LIN {X 0,Y 269.686,Z 884.674,A -85,B 0,C 180,E1 -12883.072,E2 -12883.072} C_VEL
LIN {X 0,Y 271.934,Z 878.624,A -85,B 0,C 180,E1 -12886.887,E2 -12886.887} C_VEL
LIN {X 0,Y 274.765,Z 871.156,A -85,B 0,C 180,E1 -12890.448,E2 -12890.448} C_VEL
LIN {X 0,Y 278.331,Z 861.736,A -85,B 0,C 180,E1 -12893.95,E2 -12893.95} C_VEL
LIN {X 0,Y 282.374,Z 850.757,A -85,B 0,C 180,E1 -12897.18,E2 -12897.18} C_VEL
LIN {X 0,Y 286.714,Z 838.141,A -85,B 0,C 180,E1 -12900.144,E2 -12900.144} C_VEL
LIN {X 0,Y 291.068,Z 824.299,A -85,B 0,C 180,E1 -12902.755,E2 -12902.755} C_VEL
LIN {X 0,Y 295.08,Z 810.044,A -85,B 0,C 180,E1 -12904.936,E2 -12904.936} C_VEL
LIN {X 0,Y 298.861,Z 794.399,A -85,B 0,C 180,E1 -12906.875,E2 -12906.875} C_VEL
LIN {X 0,Y 302.134,Z 778.251,A -85,B 0,C 180,E1 -12908.474,E2 -12908.474} C_VEL
LIN {X 0,Y 304.902,Z 760.982,A -85,B 0,C 180,E1 -12909.813,E2 -12909.813} C_VEL
LIN {X 0,Y 306.977,Z 742.738,A -85,B 0,C 180,E1 -12910.881,E2 -12910.881} C_VEL
LIN {X 0,Y 308.237,Z 723.755,A -85,B 0,C 180,E1 -12911.658,E2 -12911.658} C_VEL
LIN {X 0,Y 309.895,Z 682.456,A -85,B 0,C 180,E1 -12912.705,E2 -12912.705} C_VEL
LIN {X 0,Y 310.726,Z 666.212,A -85,B 0,C 180,E1 -12913.069,E2 -12913.069} C_VEL
LIN {X 0,Y 310.408,Z 658.622,A -85,B 0,C 180,E1 -12913.367,E2 -12913.367} C_VEL
LIN {X 0,Y 307.038,Z 638.78,A -85,B 0,C 180,E1 -12914.632,E2 -12914.632} C_VEL
LIN {X 0,Y 306.867,Z 632.255,A -85,B 0,C 180,E1 -12914.879,E2 -12914.879} C_VEL
LIN {X 0,Y 310.629,Z 562.408,A -85,B 0,C 180,E1 -12916.462,E2 -12916.462} C_VEL
LIN {X 0,Y 306.876,Z 565.093,A -85,B 0,C 180,E1 -12917.138,E2 -12917.138} C_VEL
LIN {X 0,Y 301.533,Z 573.563,A -85,B 0,C 180,E1 -12917.98,E2 -12917.98} C_VEL
LIN {X 0,Y 297.455,Z 578.086,A -85,B 0,C 180,E1 -12918.725,E2 -12918.725} C_VEL
LIN {X 0,Y 295.264,Z 579.155,A -85,B 0,C 180,E1 -12919.189,E2 -12919.189} C_VEL
LIN {X 0,Y 294.567,Z 579.193,A -85,B 0,C 180,E1 -12919.371,E2 -12919.371} C_VEL
LIN {X 0,Y 288.038,Z 619.211,A -85,B 0,C 180,E1 -12923.908,E2 -12923.908} C_VEL
LIN {X 0,Y 288.137,Z 629.093,A -85,B 0,C 180,E1 -12924.423,E2 -12924.423} C_VEL
LIN {X 0,Y 279.258,Z 720.889,A -85,B 0,C 180,E1 -12928.189,E2 -12928.189} C_VEL
LIN {X 0,Y 275.539,Z 766.557,A -85,B 0,C 180,E1 -12930.346,E2 -12930.346} C_VEL
LIN {X 0,Y 274.092,Z 785.081,A -85,B 0,C 180,E1 -12931.514,E2 -12931.514} C_VEL
LIN {X 0,Y 272.218,Z 802.313,A -85,B 0,C 180,E1 -12933.023,E2 -12933.023} C_VEL
LIN {X 0,Y 270.16,Z 818.126,A -85,B 0,C 180,E1 -12934.81,E2 -12934.81} C_VEL
LIN {X 0,Y 267.771,Z 834.431,A -85,B 0,C 180,E1 -12937.148,E2 -12937.148} C_VEL
LIN {X 0,Y 265.418,Z 849.249,A -85,B 0,C 180,E1 -12939.836,E2 -12939.836} C_VEL
LIN {X 0,Y 263.474,Z 861.324,A -85,B 0,C 180,E1 -12942.554,E2 -12942.554} C_VEL
LIN {X 0,Y 261.789,Z 872.401,A -85,B 0,C 180,E1 -12945.625,E2 -12945.625} C_VEL
LIN {X 0,Y 260.5,Z 881.93,A -85,B 0,C 180,E1 -12948.935,E2 -12948.935} C_VEL
LIN {X 0,Y 259.751,Z 889.559,A -85,B 0,C 180,E1 -12952.257,E2 -12952.257} C_VEL
LIN {X 0,Y 259.465,Z 896.044,A -85,B 0,C 180,E1 -12956.022,E2 -12956.022} C_VEL
LIN {X 0,Y 259.712,Z 900.395,A -85,B 0,C 180,E1 -12959.558,E2 -12959.558} C_VEL
LIN {X 0,Y 260.599,Z 903.408,A -85,B 0,C 180,E1 -12963.519,E2 -12963.519} C_VEL
LIN {X 0,Y 262.216,Z 904.421,A -85,B 0,C 180,E1 -12967.448,E2 -12967.448} C_VEL
LIN {X 0,Y 264.534,Z 903.668,A -85,B 0,C 180,E1 -12971.114,E2 -12971.114} C_VEL
LIN {X 0,Y 267.932,Z 901.106,A -85,B 0,C 180,E1 -12974.921,E2 -12974.921} C_VEL
LIN {X 0,Y 272.584,Z 896.369,A -85,B 0,C 180,E1 -12978.831,E2 -12978.831} C_VEL
LIN {X 0,Y 278.094,Z 889.924,A -85,B 0,C 180,E1 -12982.402,E2 -12982.402} C_VEL
LIN {X 0,Y 284.71,Z 881.473,A -85,B 0,C 180,E1 -12985.815,E2 -12985.815} C_VEL
LIN {X 0,Y 292.053,Z 871.644,A -85,B 0,C 180,E1 -12988.863,E2 -12988.863} C_VEL
LIN {X 0,Y 301.107,Z 859.274,A -85,B 0,C 180,E1 -12991.868,E2 -12991.868} C_VEL
LIN {X 0,Y 311.714,Z 844.887,A -85,B 0,C 180,E1 -12994.593,E2 -12994.593} C_VEL
LIN {X 0,Y 322.865,Z 830.154,A -85,B 0,C 180,E1 -12996.789,E2 -12996.789} C_VEL
LIN {X 0,Y 309.588,Z 851.693,A -85,B 0,C 180,E1 -12999.476,E2 -12999.476} C_VEL
LIN {X 0,Y 296.509,Z 873.71,A -85,B 0,C 180,E1 -13002.966,E2 -13002.966} C_VEL
LIN {X 0,Y 284.849,Z 895.114,A -85,B 0,C 180,E1 -13007.19,E2 -13007.19} C_VEL
LIN {X 0,Y 275.724,Z 913.791,A -85,B 0,C 180,E1 -13011.676,E2 -13011.676} C_VEL
LIN {X 0,Y 268.77,Z 929.861,A -85,B 0,C 180,E1 -13016.337,E2 -13016.337} C_VEL
LIN {X 0,Y 263.613,Z 943.776,A -85,B 0,C 180,E1 -13021.203,E2 -13021.203} C_VEL
LIN {X 0,Y 260.112,Z 955.453,A -85,B 0,C 180,E1 -13026.195,E2 -13026.195} C_VEL
LIN {X 0,Y 258.142,Z 964.49,A -85,B 0,C 180,E1 -13031.012,E2 -13031.012} C_VEL
LIN {X 0,Y 257.314,Z 970.99,A -85,B 0,C 180,E1 -13035.369,E2 -13035.369} C_VEL
LIN {X 0,Y 257.198,Z 975.8,A -85,B 0,C 180,E1 -13039.698,E2 -13039.698} C_VEL
LIN {X 0,Y 257.448,Z 979.006,A -85,B 0,C 180,E1 -13043.98,E2 -13043.98} C_VEL
LIN {X 0,Y 257.684,Z 980.43,A -85,B 0,C 180,E1 -13047.776,E2 -13047.776} C_VEL
LIN {X 0,Y 257.745,Z 980.427,A -85,B 0,C 180,E1 -13051.555,E2 -13051.555} C_VEL
LIN {X 0,Y 257.572,Z 979.005,A -85,B 0,C 180,E1 -13055.345,E2 -13055.345} C_VEL
LIN {X 0,Y 257.333,Z 975.954,A -85,B 0,C 180,E1 -13059.391,E2 -13059.391} C_VEL
LIN {X 0,Y 257.405,Z 971.221,A -85,B 0,C 180,E1 -13063.477,E2 -13063.477} C_VEL
LIN {X 0,Y 257.989,Z 964.85,A -85,B 0,C 180,E1 -13067.595,E2 -13067.595} C_VEL
LIN {X 0,Y 259.502,Z 955.672,A -85,B 0,C 180,E1 -13072.184,E2 -13072.184} C_VEL
LIN {X 0,Y 261.93,Z 944.738,A -85,B 0,C 180,E1 -13076.526,E2 -13076.526} C_VEL
LIN {X 0,Y 265.436,Z 931.412,A -85,B 0,C 180,E1 -13080.816,E2 -13080.816} C_VEL
LIN {X 0,Y 269.811,Z 916.263,A -85,B 0,C 180,E1 -13084.798,E2 -13084.798} C_VEL
LIN {X 0,Y 274.746,Z 899.855,A -85,B 0,C 180,E1 -13088.351,E2 -13088.351} C_VEL
LIN {X 0,Y 280.04,Z 882.42,A -85,B 0,C 180,E1 -13091.476,E2 -13091.476} C_VEL
LIN {X 0,Y 285.407,Z 864.061,A -85,B 0,C 180,E1 -13094.198,E2 -13094.198} C_VEL
LIN {X 0,Y 291.22,Z 843.632,A -85,B 0,C 180,E1 -13096.707,E2 -13096.707} C_VEL
LIN {X 0,Y 296.821,Z 822.506,A -85,B 0,C 180,E1 -13098.839,E2 -13098.839} C_VEL
LIN {X 0,Y 302.079,Z 800.854,A -85,B 0,C 180,E1 -13100.611,E2 -13100.611} C_VEL
LIN {X 0,Y 307.337,Z 776.523,A -85,B 0,C 180,E1 -13102.16,E2 -13102.16} C_VEL
LIN {X 0,Y 311.674,Z 752.148,A -85,B 0,C 180,E1 -13103.33,E2 -13103.33} C_VEL
LIN {X 0,Y 314.616,Z 728.619,A -85,B 0,C 180,E1 -13104.182,E2 -13104.182} C_VEL
LIN {X 0,Y 318.188,Z 703.693,A -85,B 0,C 180,E1 -13104.767,E2 -13104.767} C_VEL
LIN {X 0,Y 319.534,Z 697.27,A -85,B 0,C 180,E1 -13104.911,E2 -13104.911} C_VEL
LIN {X 0,Y 333.437,Z 667.218,A -85,B 0,C 180,E1 -13106.472,E2 -13106.472} C_VEL
LIN {X 0,Y 344.021,Z 646.575,A -85,B 0,C 180,E1 -13107.351,E2 -13107.351} C_VEL
LIN {X 0,Y 339.833,Z 627.474,A -85,B 0,C 180,E1 -13110.221,E2 -13110.221} C_VEL
LIN {X 0,Y 337.763,Z 606.391,A -85,B 0,C 180,E1 -13113.165,E2 -13113.165} C_VEL
LIN {X 0,Y 338.071,Z 583.429,A -85,B 0,C 180,E1 -13116.098,E2 -13116.098} C_VEL
LIN {X 0,Y 340.611,Z 559.678,A -85,B 0,C 180,E1 -13118.835,E2 -13118.835} C_VEL
LIN {X 0,Y 342.754,Z 547.466,A -85,B 0,C 180,E1 -13120.133,E2 -13120.133} C_VEL
LIN {X 0,Y 334.601,Z 531.23,A -85,B 0,C 180,E1 -13124.222,E2 -13124.222} C_VEL
LIN {X 0,Y 325.953,Z 514.792,A -85,B 0,C 180,E1 -13128.858,E2 -13128.858} C_VEL
LIN {X 0,Y 318.261,Z 500.611,A -85,B 0,C 180,E1 -13133.325,E2 -13133.325} C_VEL
LIN {X 0,Y 310.915,Z 487.26,A -85,B 0,C 180,E1 -13137.973,E2 -13137.973} C_VEL
LIN {X 0,Y 304.028,Z 475.288,A -85,B 0,C 180,E1 -13142.639,E2 -13142.639} C_VEL
LIN {X 0,Y 298.834,Z 466.349,A -85,B 0,C 180,E1 -13146.427,E2 -13146.427} C_VEL
LIN {X 0,Y 295.334,Z 460.31,A -85,B 0,C 180,E1 -13149.156,E2 -13149.156} C_VEL
LIN {X 0,Y 292.811,Z 455.963,A -85,B 0,C 180,E1 -13151.224,E2 -13151.224} C_VEL
LIN {X 0,Y 290.37,Z 451.67,A -85,B 0,C 180,E1 -13153.339,E2 -13153.339} C_VEL
LIN {X 0,Y 287.246,Z 446.365,A -85,B 0,C 180,E1 -13156.115,E2 -13156.115} C_VEL
LIN {X 0,Y 284.576,Z 441.72,A -85,B 0,C 180,E1 -13158.647,E2 -13158.647} C_VEL
LIN {X 0,Y 281.501,Z 436.433,A -85,B 0,C 180,E1 -13161.788,E2 -13161.788} C_VEL
LIN {X 0,Y 285.523,Z 436.484,A -85,B 0,C 180,E1 -13163.749,E2 -13163.749} C_VEL
LIN {X 0,Y 288.01,Z 440.52,A -85,B 0,C 180,E1 -13165.499,E2 -13165.499} C_VEL
LIN {X 0,Y 292.612,Z 448.472,A -85,B 0,C 180,E1 -13168.469,E2 -13168.469} C_VEL
LIN {X 0,Y 298.931,Z 460.913,A -85,B 0,C 180,E1 -13172.356,E2 -13172.356} C_VEL
LIN {X 0,Y 305.142,Z 474.876,A -85,B 0,C 180,E1 -13175.969,E2 -13175.969} C_VEL
LIN {X 0,Y 310.504,Z 488.843,A -85,B 0,C 180,E1 -13179.016,E2 -13179.016} C_VEL
LIN {X 0,Y 313.865,Z 499.241,A -85,B 0,C 180,E1 -13180.976,E2 -13180.976} C_VEL
LIN {X 0,Y 312.333,Z 517.888,A -85,B 0,C 180,E1 -13182.511,E2 -13182.511} C_VEL
LIN {X 0,Y 312.75,Z 525.28,A -85,B 0,C 180,E1 -13182.848,E2 -13182.848} C_VEL
LIN {X 0,Y 302.694,Z 713.065,A -85,B 0,C 180,E1 -13187.105,E2 -13187.105} C_VEL
LIN {X 0,Y 301.697,Z 734.677,A -85,B 0,C 180,E1 -13187.816,E2 -13187.816} C_VEL
LIN {X 0,Y 299.958,Z 753.181,A -85,B 0,C 180,E1 -13188.749,E2 -13188.749} C_VEL
LIN {X 0,Y 297.437,Z 770.891,A -85,B 0,C 180,E1 -13189.967,E2 -13189.967} C_VEL
LIN {X 0,Y 294.321,Z 787.313,A -85,B 0,C 180,E1 -13191.425,E2 -13191.425} C_VEL
LIN {X 0,Y 290.622,Z 803.379,A -85,B 0,C 180,E1 -13193.229,E2 -13193.229} C_VEL
LIN {X 0,Y 286.527,Z 818.441,A -85,B 0,C 180,E1 -13195.334,E2 -13195.334} C_VEL
LIN {X 0,Y 282.137,Z 832.541,A -85,B 0,C 180,E1 -13197.768,E2 -13197.768} C_VEL
LIN {X 0,Y 277.8,Z 845.153,A -85,B 0,C 180,E1 -13200.457,E2 -13200.457} C_VEL
LIN {X 0,Y 273.502,Z 856.753,A -85,B 0,C 180,E1 -13203.513,E2 -13203.513} C_VEL
LIN {X 0,Y 269.379,Z 867.277,A -85,B 0,C 180,E1 -13207.002,E2 -13207.002} C_VEL
LIN {X 0,Y 265.876,Z 876.028,A -85,B 0,C 180,E1 -13210.722,E2 -13210.722} C_VEL
LIN {X 0,Y 263.109,Z 882.968,A -85,B 0,C 180,E1 -13214.574,E2 -13214.574} C_VEL
LIN {X 0,Y 261.045,Z 888.364,A -85,B 0,C 180,E1 -13218.679,E2 -13218.679} C_VEL
LIN {X 0,Y 259.745,Z 892.055,A -85,B 0,C 180,E1 -13222.925,E2 -13222.925} C_VEL
LIN {X 0,Y 259.111,Z 893.998,A -85,B 0,C 180,E1 -13227.125,E2 -13227.125} C_VEL
LIN {X 0,Y 259.011,Z 894.319,A -85,B 0,C 180,E1 -13231.328,E2 -13231.328} C_VEL
LIN {X 0,Y 259.438,Z 893.029,A -85,B 0,C 180,E1 -13235.53,E2 -13235.53} C_VEL
LIN {X 0,Y 260.445,Z 890.085,A -85,B 0,C 180,E1 -13239.726,E2 -13239.726} C_VEL
LIN {X 0,Y 262.204,Z 885.377,A -85,B 0,C 180,E1 -13243.901,E2 -13243.901} C_VEL
LIN {X 0,Y 264.702,Z 879.086,A -85,B 0,C 180,E1 -13247.845,E2 -13247.845} C_VEL
LIN {X 0,Y 267.966,Z 870.939,A -85,B 0,C 180,E1 -13251.679,E2 -13251.679} C_VEL
LIN {X 0,Y 271.854,Z 861.1,A -85,B 0,C 180,E1 -13255.255,E2 -13255.255} C_VEL
LIN {X 0,Y 275.924,Z 850.446,A -85,B 0,C 180,E1 -13258.341,E2 -13258.341} C_VEL
LIN {X 0,Y 280.217,Z 838.43,A -85,B 0,C 180,E1 -13261.158,E2 -13261.158} C_VEL
LIN {X 0,Y 284.623,Z 824.969,A -85,B 0,C 180,E1 -13263.714,E2 -13263.714} C_VEL
LIN {X 0,Y 288.821,Z 810.587,A -85,B 0,C 180,E1 -13265.93,E2 -13265.93} C_VEL
LIN {X 0,Y 292.63,Z 795.395,A -85,B 0,C 180,E1 -13267.83,E2 -13267.83} C_VEL
LIN {X 0,Y 295.986,Z 779.481,A -85,B 0,C 180,E1 -13269.426,E2 -13269.426} C_VEL
LIN {X 0,Y 298.869,Z 762.198,A -85,B 0,C 180,E1 -13270.784,E2 -13270.784} C_VEL
LIN {X 0,Y 301.034,Z 743.929,A -85,B 0,C 180,E1 -13271.867,E2 -13271.867} C_VEL
LIN {X 0,Y 302.358,Z 724.895,A -85,B 0,C 180,E1 -13272.657,E2 -13272.657} C_VEL
LIN {X 0,Y 304.093,Z 683.595,A -85,B 0,C 180,E1 -13273.721,E2 -13273.721} C_VEL
LIN {X 0,Y 306.867,Z 632.255,A -85,B 0,C 180,E1 -13274.879,E2 -13274.879} C_VEL
LIN {X 0,Y 306.592,Z 624.667,A -85,B 0,C 180,E1 -13275.183,E2 -13275.183} C_VEL
LIN {X 0,Y 303.427,Z 604.831,A -85,B 0,C 180,E1 -13276.486,E2 -13276.486} C_VEL
LIN {X 0,Y 303.291,Z 598.308,A -85,B 0,C 180,E1 -13276.739,E2 -13276.739} C_VEL
LIN {X 0,Y 304.281,Z 579.807,A -85,B 0,C 180,E1 -13277.172,E2 -13277.172} C_VEL
LIN {X 0,Y 299.607,Z 584.811,A -85,B 0,C 180,E1 -13278,E2 -13278} C_VEL
LIN {X 0,Y 296.722,Z 586.907,A -85,B 0,C 180,E1 -13278.568,E2 -13278.568} C_VEL
LIN {X 0,Y 291.301,Z 595.969,A -85,B 0,C 180,E1 -13279.489,E2 -13279.489} C_VEL
LIN {X 0,Y 287.307,Z 600.801,A -85,B 0,C 180,E1 -13280.274,E2 -13280.274} C_VEL
LIN {X 0,Y 284.901,Z 602.253,A -85,B 0,C 180,E1 -13280.823,E2 -13280.823} C_VEL
LIN {X 0,Y 284.207,Z 602.229,A -85,B 0,C 180,E1 -13281.011,E2 -13281.011} C_VEL
LIN {X 0,Y 281.343,Z 620.048,A -85,B 0,C 180,E1 -13283.037,E2 -13283.037} C_VEL
LIN {X 0,Y 281.385,Z 629.859,A -85,B 0,C 180,E1 -13283.565,E2 -13283.565} C_VEL
LIN {X 0,Y 271.871,Z 723.942,A -85,B 0,C 180,E1 -13287.555,E2 -13287.555} C_VEL
LIN {X 0,Y 268.167,Z 767.49,A -85,B 0,C 180,E1 -13289.708,E2 -13289.708} C_VEL
LIN {X 0,Y 266.603,Z 786.293,A -85,B 0,C 180,E1 -13290.943,E2 -13290.943} C_VEL
LIN {X 0,Y 264.596,Z 804.008,A -85,B 0,C 180,E1 -13292.547,E2 -13292.547} C_VEL
LIN {X 0,Y 262.469,Z 819.69,A -85,B 0,C 180,E1 -13294.381,E2 -13294.381} C_VEL
LIN {X 0,Y 260.11,Z 835.238,A -85,B 0,C 180,E1 -13296.675,E2 -13296.675} C_VEL
LIN {X 0,Y 257.753,Z 849.521,A -85,B 0,C 180,E1 -13299.328,E2 -13299.328} C_VEL
LIN {X 0,Y 255.647,Z 862.213,A -85,B 0,C 180,E1 -13302.237,E2 -13302.237} C_VEL
LIN {X 0,Y 253.798,Z 874.116,A -85,B 0,C 180,E1 -13305.629,E2 -13305.629} C_VEL
LIN {X 0,Y 252.446,Z 884.164,A -85,B 0,C 180,E1 -13309.271,E2 -13309.271} C_VEL
LIN {X 0,Y 251.737,Z 891.577,A -85,B 0,C 180,E1 -13312.697,E2 -13312.697} C_VEL
LIN {X 0,Y 251.545,Z 897.997,A -85,B 0,C 180,E1 -13316.581,E2 -13316.581} C_VEL
LIN {X 0,Y 251.945,Z 902.424,A -85,B 0,C 180,E1 -13320.454,E2 -13320.454} C_VEL
LIN {X 0,Y 252.97,Z 905.133,A -85,B 0,C 180,E1 -13324.306,E2 -13324.306} C_VEL
LIN {X 0,Y 254.835,Z 906.14,A -85,B 0,C 180,E1 -13328.347,E2 -13328.347} C_VEL
LIN {X 0,Y 257.823,Z 905.177,A -85,B 0,C 180,E1 -13332.542,E2 -13332.542} C_VEL
LIN {X 0,Y 261.946,Z 902.204,A -85,B 0,C 180,E1 -13336.635,E2 -13336.635} C_VEL
LIN {X 0,Y 267.259,Z 897.237,A -85,B 0,C 180,E1 -13340.589,E2 -13340.589} C_VEL
LIN {X 0,Y 273.829,Z 890.233,A -85,B 0,C 180,E1 -13344.368,E2 -13344.368} C_VEL
LIN {X 0,Y 281.246,Z 881.626,A -85,B 0,C 180,E1 -13347.756,E2 -13347.756} C_VEL
LIN {X 0,Y 290.467,Z 870.573,A -85,B 0,C 180,E1 -13351.086,E2 -13351.086} C_VEL
LIN {X 0,Y 301.272,Z 857.503,A -85,B 0,C 180,E1 -13354.116,E2 -13354.116} C_VEL
LIN {X 0,Y 313.457,Z 843.065,A -85,B 0,C 180,E1 -13356.732,E2 -13356.732} C_VEL
LIN {X 0,Y 299.81,Z 863.023,A -85,B 0,C 180,E1 -13359.611,E2 -13359.611} C_VEL
LIN {X 0,Y 286.869,Z 883.051,A -85,B 0,C 180,E1 -13363.242,E2 -13363.242} C_VEL
LIN {X 0,Y 275.073,Z 903.185,A -85,B 0,C 180,E1 -13367.742,E2 -13367.742} C_VEL
LIN {X 0,Y 265.677,Z 921.336,A -85,B 0,C 180,E1 -13372.705,E2 -13372.705} C_VEL
LIN {X 0,Y 258.843,Z 936.59,A -85,B 0,C 180,E1 -13377.786,E2 -13377.786} C_VEL
LIN {X 0,Y 253.997,Z 949.606,A -85,B 0,C 180,E1 -13383.082,E2 -13383.082} C_VEL
LIN {X 0,Y 250.974,Z 960.274,A -85,B 0,C 180,E1 -13388.498,E2 -13388.498} C_VEL
LIN {X 0,Y 249.639,Z 967.637,A -85,B 0,C 180,E1 -13393.239,E2 -13393.239} C_VEL
LIN {X 0,Y 249.22,Z 973.262,A -85,B 0,C 180,E1 -13397.958,E2 -13397.958} C_VEL
LIN {X 0,Y 249.399,Z 976.902,A -85,B 0,C 180,E1 -13402.397,E2 -13402.397} C_VEL
LIN {X 0,Y 249.717,Z 978.754,A -85,B 0,C 180,E1 -13406.326,E2 -13406.326} C_VEL
LIN {X 0,Y 249.877,Z 979.213,A -85,B 0,C 180,E1 -13410.229,E2 -13410.229} C_VEL
LIN {X 0,Y 249.769,Z 978.324,A -85,B 0,C 180,E1 -13413.902,E2 -13413.902} C_VEL
LIN {X 0,Y 249.523,Z 975.953,A -85,B 0,C 180,E1 -13417.83,E2 -13417.83} C_VEL
LIN {X 0,Y 249.426,Z 971.821,A -85,B 0,C 180,E1 -13422.031,E2 -13422.031} C_VEL
LIN {X 0,Y 249.806,Z 966.033,A -85,B 0,C 180,E1 -13426.27,E2 -13426.27} C_VEL
LIN {X 0,Y 250.953,Z 958.015,A -85,B 0,C 180,E1 -13430.768,E2 -13430.768} C_VEL
LIN {X 0,Y 253.071,Z 947.881,A -85,B 0,C 180,E1 -13435.257,E2 -13435.257} C_VEL
LIN {X 0,Y 256.087,Z 936.144,A -85,B 0,C 180,E1 -13439.468,E2 -13439.468} C_VEL
LIN {X 0,Y 259.96,Z 922.745,A -85,B 0,C 180,E1 -13443.424,E2 -13443.424} C_VEL
LIN {X 0,Y 264.675,Z 907.329,A -85,B 0,C 180,E1 -13447.187,E2 -13447.187} C_VEL
LIN {X 0,Y 270.058,Z 890.071,A -85,B 0,C 180,E1 -13450.663,E2 -13450.663} C_VEL
LIN {X 0,Y 275.908,Z 871.132,A -85,B 0,C 180,E1 -13453.801,E2 -13453.801} C_VEL
LIN {X 0,Y 281.61,Z 851.907,A -85,B 0,C 180,E1 -13456.41,E2 -13456.41} C_VEL
LIN {X 0,Y 287.648,Z 830.425,A -85,B 0,C 180,E1 -13458.811,E2 -13458.811} C_VEL
LIN {X 0,Y 293.436,Z 808.148,A -85,B 0,C 180,E1 -13460.821,E2 -13460.821} C_VEL
LIN {X 0,Y 298.595,Z 785.998,A -85,B 0,C 180,E1 -13462.417,E2 -13462.417} C_VEL
LIN {X 0,Y 303.411,Z 762.358,A -85,B 0,C 180,E1 -13463.729,E2 -13463.729} C_VEL
LIN {X 0,Y 307.137,Z 738.225,A -85,B 0,C 180,E1 -13464.751,E2 -13464.751} C_VEL
LIN {X 0,Y 310.167,Z 714.56,A -85,B 0,C 180,E1 -13465.45,E2 -13465.45} C_VEL
LIN {X 0,Y 313.131,Z 697.099,A -85,B 0,C 180,E1 -13465.792,E2 -13465.792} C_VEL
LIN {X 0,Y 326.242,Z 669.122,A -85,B 0,C 180,E1 -13467.275,E2 -13467.275} C_VEL
LIN {X 0,Y 336.947,Z 647.982,A -85,B 0,C 180,E1 -13468.214,E2 -13468.214} C_VEL
LIN {X 0,Y 333.158,Z 628.831,A -85,B 0,C 180,E1 -13471.107,E2 -13471.107} C_VEL
LIN {X 0,Y 331.41,Z 607.06,A -85,B 0,C 180,E1 -13474.155,E2 -13474.155} C_VEL
LIN {X 0,Y 332.113,Z 583.658,A -85,B 0,C 180,E1 -13477.148,E2 -13477.148} C_VEL
LIN {X 0,Y 335.13,Z 559.549,A -85,B 0,C 180,E1 -13479.935,E2 -13479.935} C_VEL
LIN {X 0,Y 336.475,Z 551.398,A -85,B 0,C 180,E1 -13480.831,E2 -13480.831} C_VEL
LIN {X 0,Y 328.678,Z 535.801,A -85,B 0,C 180,E1 -13484.834,E2 -13484.834} C_VEL
LIN {X 0,Y 320.059,Z 519.312,A -85,B 0,C 180,E1 -13489.561,E2 -13489.561} C_VEL
LIN {X 0,Y 312.61,Z 505.626,A -85,B 0,C 180,E1 -13493.942,E2 -13493.942} C_VEL
LIN {X 0,Y 305.813,Z 493.164,A -85,B 0,C 180,E1 -13498.314,E2 -13498.314} C_VEL
LIN {X 0,Y 299.308,Z 481.764,A -85,B 0,C 180,E1 -13502.781,E2 -13502.781} C_VEL
LIN {X 0,Y 293.979,Z 472.523,A -85,B 0,C 180,E1 -13506.725,E2 -13506.725} C_VEL
LIN {X 0,Y 289.311,Z 464.05,A -85,B 0,C 180,E1 -13510.555,E2 -13510.555} C_VEL
LIN {X 0,Y 285.153,Z 457.26,A -85,B 0,C 180,E1 -13514.002,E2 -13514.002} C_VEL
LIN {X 0,Y 282.474,Z 452.599,A -85,B 0,C 180,E1 -13516.45,E2 -13516.45} C_VEL
LIN {X 0,Y 279.859,Z 448.022,A -85,B 0,C 180,E1 -13518.973,E2 -13518.973} C_VEL
LIN {X 0,Y 277.749,Z 444.16,A -85,B 0,C 180,E1 -13521.249,E2 -13521.249} C_VEL
LIN {X 0,Y 282.462,Z 444.013,A -85,B 0,C 180,E1 -13523.579,E2 -13523.579} C_VEL
LIN {X 0,Y 284.896,Z 448.146,A -85,B 0,C 180,E1 -13525.352,E2 -13525.352} C_VEL
LIN {X 0,Y 288.855,Z 455.355,A -85,B 0,C 180,E1 -13528.084,E2 -13528.084} C_VEL
LIN {X 0,Y 294.565,Z 466.832,A -85,B 0,C 180,E1 -13531.745,E2 -13531.745} C_VEL
LIN {X 0,Y 300.575,Z 480.76,A -85,B 0,C 180,E1 -13535.415,E2 -13535.415} C_VEL
LIN {X 0,Y 305.795,Z 494.827,A -85,B 0,C 180,E1 -13538.527,E2 -13538.527} C_VEL
LIN {X 0,Y 308.386,Z 502.912,A -85,B 0,C 180,E1 -13540.079,E2 -13540.079} C_VEL
LIN {X 0,Y 307.017,Z 519.225,A -85,B 0,C 180,E1 -13541.424,E2 -13541.424} C_VEL
LIN {X 0,Y 307.393,Z 526.483,A -85,B 0,C 180,E1 -13541.762,E2 -13541.762} C_VEL
LIN {X 0,Y 296.955,Z 713.471,A -85,B 0,C 180,E1 -13546.042,E2 -13546.042} C_VEL
LIN {X 0,Y 295.929,Z 735.122,A -85,B 0,C 180,E1 -13546.754,E2 -13546.754} C_VEL
LIN {X 0,Y 294.106,Z 753.997,A -85,B 0,C 180,E1 -13547.708,E2 -13547.708} C_VEL
LIN {X 0,Y 291.534,Z 771.501,A -85,B 0,C 180,E1 -13548.918,E2 -13548.918} C_VEL
LIN {X 0,Y 288.165,Z 788.657,A -85,B 0,C 180,E1 -13550.455,E2 -13550.455} C_VEL
LIN {X 0,Y 284.23,Z 805.042,A -85,B 0,C 180,E1 -13552.327,E2 -13552.327} C_VEL
LIN {X 0,Y 280.062,Z 819.698,A -85,B 0,C 180,E1 -13554.414,E2 -13554.414} C_VEL
LIN {X 0,Y 275.479,Z 833.801,A -85,B 0,C 180,E1 -13556.891,E2 -13556.891} C_VEL
LIN {X 0,Y 270.943,Z 846.416,A -85,B 0,C 180,E1 -13559.631,E2 -13559.631} C_VEL
LIN {X 0,Y 266.308,Z 858.348,A -85,B 0,C 180,E1 -13562.852,E2 -13562.852} C_VEL
LIN {X 0,Y 262.04,Z 868.686,A -85,B 0,C 180,E1 -13566.382,E2 -13566.382} C_VEL
LIN {X 0,Y 258.446,Z 877.208,A -85,B 0,C 180,E1 -13570.096,E2 -13570.096} C_VEL
LIN {X 0,Y 255.48,Z 884.235,A -85,B 0,C 180,E1 -13574.101,E2 -13574.101} C_VEL
LIN {X 0,Y 253.354,Z 889.462,A -85,B 0,C 180,E1 -13578.164,E2 -13578.164} C_VEL
LIN {X 0,Y 251.95,Z 893.175,A -85,B 0,C 180,E1 -13582.476,E2 -13582.476} C_VEL
LIN {X 0,Y 251.24,Z 895.199,A -85,B 0,C 180,E1 -13586.807,E2 -13586.807} C_VEL
LIN {X 0,Y 251.107,Z 895.602,A -85,B 0,C 180,E1 -13591.141,E2 -13591.141} C_VEL
LIN {X 0,Y 251.529,Z 894.396,A -85,B 0,C 180,E1 -13595.475,E2 -13595.475} C_VEL
LIN {X 0,Y 252.57,Z 891.54,A -85,B 0,C 180,E1 -13599.802,E2 -13599.802} C_VEL
LIN {X 0,Y 254.278,Z 887.204,A -85,B 0,C 180,E1 -13603.879,E2 -13603.879} C_VEL
LIN {X 0,Y 256.807,Z 881.153,A -85,B 0,C 180,E1 -13607.914,E2 -13607.914} C_VEL
LIN {X 0,Y 259.97,Z 873.683,A -85,B 0,C 180,E1 -13611.668,E2 -13611.668} C_VEL
LIN {X 0,Y 263.928,Z 864.259,A -85,B 0,C 180,E1 -13615.347,E2 -13615.347} C_VEL
LIN {X 0,Y 268.384,Z 853.274,A -85,B 0,C 180,E1 -13618.725,E2 -13618.725} C_VEL
LIN {X 0,Y 273.144,Z 840.65,A -85,B 0,C 180,E1 -13621.812,E2 -13621.812} C_VEL
LIN {X 0,Y 277.898,Z 826.8,A -85,B 0,C 180,E1 -13624.519,E2 -13624.519} C_VEL
LIN {X 0,Y 282.265,Z 812.534,A -85,B 0,C 180,E1 -13626.774,E2 -13626.774} C_VEL
LIN {X 0,Y 286.429,Z 796.633,A -85,B 0,C 180,E1 -13628.8,E2 -13628.8} C_VEL
LIN {X 0,Y 289.924,Z 780.711,A -85,B 0,C 180,E1 -13630.419,E2 -13630.419} C_VEL
LIN {X 0,Y 292.927,Z 763.415,A -85,B 0,C 180,E1 -13631.795,E2 -13631.795} C_VEL
LIN {X 0,Y 295.185,Z 745.123,A -85,B 0,C 180,E1 -13632.893,E2 -13632.893} C_VEL
LIN {X 0,Y 296.584,Z 725.841,A -85,B 0,C 180,E1 -13633.702,E2 -13633.702} C_VEL
LIN {X 0,Y 298.419,Z 684.225,A -85,B 0,C 180,E1 -13634.788,E2 -13634.788} C_VEL
LIN {X 0,Y 303.291,Z 598.308,A -85,B 0,C 180,E1 -13636.739,E2 -13636.739} C_VEL
LIN {X 0,Y 302.549,Z 597.158,A -85,B 0,C 180,E1 -13636.933,E2 -13636.933} C_VEL
LIN {X 0,Y 300.704,Z 597.207,A -85,B 0,C 180,E1 -13637.322,E2 -13637.322} C_VEL
LIN {X 0,Y 297.682,Z 599.077,A -85,B 0,C 180,E1 -13637.912,E2 -13637.912} C_VEL
LIN {X 0,Y 288.788,Z 608.027,A -85,B 0,C 180,E1 -13639.631,E2 -13639.631} C_VEL
LIN {X 0,Y 288.17,Z 608.506,A -85,B 0,C 180,E1 -13639.763,E2 -13639.763} C_VEL
LIN {X 0,Y 286.362,Z 609.844,A -85,B 0,C 180,E1 -13640.155,E2 -13640.155} C_VEL
LIN {X 0,Y 280.676,Z 619.876,A -85,B 0,C 180,E1 -13641.205,E2 -13641.205} C_VEL
LIN {X 0,Y 276.484,Z 626.349,A -85,B 0,C 180,E1 -13642.064,E2 -13642.064} C_VEL
LIN {X 0,Y 274.919,Z 627.057,A -85,B 0,C 180,E1 -13642.469,E2 -13642.469} C_VEL
LIN {X 0,Y 274.299,Z 633.934,A -85,B 0,C 180,E1 -13642.813,E2 -13642.813} C_VEL
LIN {X 0,Y 265.197,Z 720.212,A -85,B 0,C 180,E1 -13646.577,E2 -13646.577} C_VEL
LIN {X 0,Y 260.999,Z 765.773,A -85,B 0,C 180,E1 -13648.897,E2 -13648.897} C_VEL
LIN {X 0,Y 259.479,Z 784.13,A -85,B 0,C 180,E1 -13650.078,E2 -13650.078} C_VEL
LIN {X 0,Y 257.535,Z 801.508,A -85,B 0,C 180,E1 -13651.601,E2 -13651.601} C_VEL
LIN {X 0,Y 255.165,Z 818.62,A -85,B 0,C 180,E1 -13653.592,E2 -13653.592} C_VEL
LIN {X 0,Y 252.786,Z 833.799,A -85,B 0,C 180,E1 -13655.833,E2 -13655.833} C_VEL
LIN {X 0,Y 250.392,Z 848.104,A -85,B 0,C 180,E1 -13658.446,E2 -13658.446} C_VEL
LIN {X 0,Y 247.98,Z 862.215,A -85,B 0,C 180,E1 -13661.669,E2 -13661.669} C_VEL
LIN {X 0,Y 246.125,Z 873.574,A -85,B 0,C 180,E1 -13664.93,E2 -13664.93} C_VEL
LIN {X 0,Y 244.719,Z 883.474,A -85,B 0,C 180,E1 -13668.451,E2 -13668.451} C_VEL
LIN {X 0,Y 243.828,Z 892.315,A -85,B 0,C 180,E1 -13672.459,E2 -13672.459} C_VEL
LIN {X 0,Y 243.608,Z 898.897,A -85,B 0,C 180,E1 -13676.47,E2 -13676.47} C_VEL
LIN {X 0,Y 243.997,Z 903.382,A -85,B 0,C 180,E1 -13680.234,E2 -13680.234} C_VEL
LIN {X 0,Y 245.121,Z 906.563,A -85,B 0,C 180,E1 -13684.444,E2 -13684.444} C_VEL
LIN {X 0,Y 247.093,Z 907.799,A -85,B 0,C 180,E1 -13688.61,E2 -13688.61} C_VEL
LIN {X 0,Y 249.92,Z 907.305,A -85,B 0,C 180,E1 -13692.529,E2 -13692.529} C_VEL
LIN {X 0,Y 253.866,Z 905.131,A -85,B 0,C 180,E1 -13696.473,E2 -13696.473} C_VEL
LIN {X 0,Y 259.27,Z 900.897,A -85,B 0,C 180,E1 -13700.544,E2 -13700.544} C_VEL
LIN {X 0,Y 265.968,Z 894.7,A -85,B 0,C 180,E1 -13704.426,E2 -13704.426} C_VEL
LIN {X 0,Y 274.02,Z 886.578,A -85,B 0,C 180,E1 -13708.079,E2 -13708.079} C_VEL
LIN {X 0,Y 283.489,Z 876.532,A -85,B 0,C 180,E1 -13711.465,E2 -13711.465} C_VEL
LIN {X 0,Y 294.535,Z 864.684,A -85,B 0,C 180,E1 -13714.535,E2 -13714.535} C_VEL
LIN {X 0,Y 304.084,Z 854.614,A -85,B 0,C 180,E1 -13716.649,E2 -13716.649} C_VEL
LIN {X 0,Y 289.382,Z 874.155,A -85,B 0,C 180,E1 -13719.91,E2 -13719.91} C_VEL
LIN {X 0,Y 275.619,Z 894.001,A -85,B 0,C 180,E1 -13724.086,E2 -13724.086} C_VEL
LIN {X 0,Y 264.226,Z 912.38,A -85,B 0,C 180,E1 -13728.853,E2 -13728.853} C_VEL
LIN {X 0,Y 255.373,Z 928.759,A -85,B 0,C 180,E1 -13734.034,E2 -13734.034} C_VEL
LIN {X 0,Y 248.816,Z 943.067,A -85,B 0,C 180,E1 -13739.58,E2 -13739.58} C_VEL
LIN {X 0,Y 244.46,Z 955.034,A -85,B 0,C 180,E1 -13745.342,E2 -13745.342} C_VEL
LIN {X 0,Y 242.201,Z 963.833,A -85,B 0,C 180,E1 -13750.715,E2 -13750.715} C_VEL
LIN {X 0,Y 241.342,Z 970.047,A -85,B 0,C 180,E1 -13755.606,E2 -13755.606} C_VEL
LIN {X 0,Y 241.327,Z 974.467,A -85,B 0,C 180,E1 -13760.423,E2 -13760.423} C_VEL
LIN {X 0,Y 241.695,Z 976.968,A -85,B 0,C 180,E1 -13764.778,E2 -13764.778} C_VEL
LIN {X 0,Y 241.949,Z 977.845,A -85,B 0,C 180,E1 -13768.579,E2 -13768.579} C_VEL
LIN {X 0,Y 241.961,Z 977.426,A -85,B 0,C 180,E1 -13772.368,E2 -13772.368} C_VEL
LIN {X 0,Y 241.741,Z 975.693,A -85,B 0,C 180,E1 -13776.173,E2 -13776.173} C_VEL
LIN {X 0,Y 241.533,Z 972.176,A -85,B 0,C 180,E1 -13780.494,E2 -13780.494} C_VEL
LIN {X 0,Y 241.685,Z 966.958,A -85,B 0,C 180,E1 -13784.862,E2 -13784.862} C_VEL
LIN {X 0,Y 242.585,Z 959.581,A -85,B 0,C 180,E1 -13789.502,E2 -13789.502} C_VEL
LIN {X 0,Y 244.478,Z 949.952,A -85,B 0,C 180,E1 -13794.216,E2 -13794.216} C_VEL
LIN {X 0,Y 247.405,Z 938.395,A -85,B 0,C 180,E1 -13798.745,E2 -13798.745} C_VEL
LIN {X 0,Y 251.317,Z 924.96,A -85,B 0,C 180,E1 -13803.028,E2 -13803.028} C_VEL
LIN {X 0,Y 256.337,Z 908.901,A -85,B 0,C 180,E1 -13807.198,E2 -13807.198} C_VEL
LIN {X 0,Y 261.759,Z 892.042,A -85,B 0,C 180,E1 -13810.781,E2 -13810.781} C_VEL
LIN {X 0,Y 267.653,Z 873.543,A -85,B 0,C 180,E1 -13814.013,E2 -13814.013} C_VEL
LIN {X 0,Y 274.081,Z 852.614,A -85,B 0,C 180,E1 -13816.986,E2 -13816.986} C_VEL
LIN {X 0,Y 280.27,Z 831.368,A -85,B 0,C 180,E1 -13819.452,E2 -13819.452} C_VEL
LIN {X 0,Y 286.024,Z 810.155,A -85,B 0,C 180,E1 -13821.453,E2 -13821.453} C_VEL
LIN {X 0,Y 291.623,Z 787.095,A -85,B 0,C 180,E1 -13823.185,E2 -13823.185} C_VEL
LIN {X 0,Y 296.558,Z 763.743,A -85,B 0,C 180,E1 -13824.528,E2 -13824.528} C_VEL
LIN {X 0,Y 300.375,Z 740.597,A -85,B 0,C 180,E1 -13825.554,E2 -13825.554} C_VEL
LIN {X 0,Y 303.532,Z 716.707,A -85,B 0,C 180,E1 -13826.317,E2 -13826.317} C_VEL
LIN {X 0,Y 307.211,Z 695.979,A -85,B 0,C 180,E1 -13826.765,E2 -13826.765} C_VEL
LIN {X 0,Y 320.891,Z 667.189,A -85,B 0,C 180,E1 -13828.28,E2 -13828.28} C_VEL
LIN {X 0,Y 329.956,Z 649.505,A -85,B 0,C 180,E1 -13829.069,E2 -13829.069} C_VEL
LIN {X 0,Y 326.455,Z 629.792,A -85,B 0,C 180,E1 -13832.057,E2 -13832.057} C_VEL
LIN {X 0,Y 325.123,Z 607.674,A -85,B 0,C 180,E1 -13835.17,E2 -13835.17} C_VEL
LIN {X 0,Y 326.266,Z 583.81,A -85,B 0,C 180,E1 -13838.235,E2 -13838.235} C_VEL
LIN {X 0,Y 329.725,Z 559.257,A -85,B 0,C 180,E1 -13841.067,E2 -13841.067} C_VEL
LIN {X 0,Y 330.361,Z 555.633,A -85,B 0,C 180,E1 -13841.471,E2 -13841.471} C_VEL
LIN {X 0,Y 322.393,Z 539.664,A -85,B 0,C 180,E1 -13845.635,E2 -13845.635} C_VEL
LIN {X 0,Y 314.37,Z 524.322,A -85,B 0,C 180,E1 -13850.111,E2 -13850.111} C_VEL
LIN {X 0,Y 307.27,Z 511.131,A -85,B 0,C 180,E1 -13854.398,E2 -13854.398} C_VEL
LIN {X 0,Y 300.705,Z 499.055,A -85,B 0,C 180,E1 -13858.667,E2 -13858.667} C_VEL
LIN {X 0,Y 294.032,Z 487.282,A -85,B 0,C 180,E1 -13863.315,E2 -13863.315} C_VEL
LIN {X 0,Y 288.963,Z 478.427,A -85,B 0,C 180,E1 -13867.156,E2 -13867.156} C_VEL
LIN {X 0,Y 284.226,Z 469.919,A -85,B 0,C 180,E1 -13871.048,E2 -13871.048} C_VEL
LIN {X 0,Y 280.493,Z 463.656,A -85,B 0,C 180,E1 -13874.239,E2 -13874.239} C_VEL
LIN {X 0,Y 277.756,Z 458.895,A -85,B 0,C 180,E1 -13876.758,E2 -13876.758} C_VEL
LIN {X 0,Y 275.136,Z 454.308,A -85,B 0,C 180,E1 -13879.312,E2 -13879.312} C_VEL
LIN {X 0,Y 273.857,Z 452.2,A -85,B 0,C 180,E1 -13880.63,E2 -13880.63} C_VEL
LIN {X 0,Y 278.192,Z 451.69,A -85,B 0,C 180,E1 -13882.841,E2 -13882.841} C_VEL
LIN {X 0,Y 279.655,Z 451.933,A -85,B 0,C 180,E1 -13883.606,E2 -13883.606} C_VEL
LIN {X 0,Y 283.32,Z 458.734,A -85,B 0,C 180,E1 -13886.402,E2 -13886.402} C_VEL
LIN {X 0,Y 288.788,Z 469.567,A -85,B 0,C 180,E1 -13890.135,E2 -13890.135} C_VEL
LIN {X 0,Y 294.094,Z 481.798,A -85,B 0,C 180,E1 -13893.598,E2 -13893.598} C_VEL
LIN {X 0,Y 298.932,Z 494.276,A -85,B 0,C 180,E1 -13896.608,E2 -13896.608} C_VEL
LIN {X 0,Y 302.985,Z 506.585,A -85,B 0,C 180,E1 -13899.15,E2 -13899.15} C_VEL
LIN {X 0,Y 301.799,Z 520.344,A -85,B 0,C 180,E1 -13900.287,E2 -13900.287} C_VEL
LIN {X 0,Y 302.153,Z 527.661,A -85,B 0,C 180,E1 -13900.638,E2 -13900.638} C_VEL
LIN {X 0,Y 291.318,Z 714.004,A -85,B 0,C 180,E1 -13904.942,E2 -13904.942} C_VEL
LIN {X 0,Y 290.256,Z 735.722,A -85,B 0,C 180,E1 -13905.657,E2 -13905.657} C_VEL
LIN {X 0,Y 288.342,Z 754.919,A -85,B 0,C 180,E1 -13906.632,E2 -13906.632} C_VEL
LIN {X 0,Y 285.674,Z 772.454,A -85,B 0,C 180,E1 -13907.853,E2 -13907.853} C_VEL
LIN {X 0,Y 282.116,Z 789.905,A -85,B 0,C 180,E1 -13909.433,E2 -13909.433} C_VEL
LIN {X 0,Y 278.123,Z 805.885,A -85,B 0,C 180,E1 -13911.279,E2 -13911.279} C_VEL
LIN {X 0,Y 273.672,Z 820.954,A -85,B 0,C 180,E1 -13913.451,E2 -13913.451} C_VEL
LIN {X 0,Y 268.889,Z 835.061,A -85,B 0,C 180,E1 -13915.97,E2 -13915.97} C_VEL
LIN {X 0,Y 263.974,Z 848.141,A -85,B 0,C 180,E1 -13918.874,E2 -13918.874} C_VEL
LIN {X 0,Y 259.129,Z 859.973,A -85,B 0,C 180,E1 -13922.168,E2 -13922.168} C_VEL
LIN {X 0,Y 254.799,Z 869.953,A -85,B 0,C 180,E1 -13925.668,E2 -13925.668} C_VEL
LIN {X 0,Y 251.008,Z 878.475,A -85,B 0,C 180,E1 -13929.48,E2 -13929.48} C_VEL
LIN {X 0,Y 247.87,Z 885.502,A -85,B 0,C 180,E1 -13933.599,E2 -13933.599} C_VEL
LIN {X 0,Y 245.611,Z 890.723,A -85,B 0,C 180,E1 -13937.779,E2 -13937.779} C_VEL
LIN {X 0,Y 244.11,Z 894.44,A -85,B 0,C 180,E1 -13942.232,E2 -13942.232} C_VEL
LIN {X 0,Y 243.338,Z 896.499,A -85,B 0,C 180,E1 -13946.841,E2 -13946.841} C_VEL
LIN {X 0,Y 243.215,Z 896.846,A -85,B 0,C 180,E1 -13951.414,E2 -13951.414} C_VEL
LIN {X 0,Y 243.703,Z 895.557,A -85,B 0,C 180,E1 -13955.888,E2 -13955.888} C_VEL
LIN {X 0,Y 244.855,Z 892.615,A -85,B 0,C 180,E1 -13960.351,E2 -13960.351} C_VEL
LIN {X 0,Y 246.852,Z 887.908,A -85,B 0,C 180,E1 -13964.785,E2 -13964.785} C_VEL
LIN {X 0,Y 249.636,Z 881.662,A -85,B 0,C 180,E1 -13968.932,E2 -13968.932} C_VEL
LIN {X 0,Y 253.302,Z 873.466,A -85,B 0,C 180,E1 -13973.004,E2 -13973.004} C_VEL
LIN {X 0,Y 257.612,Z 863.621,A -85,B 0,C 180,E1 -13976.759,E2 -13976.759} C_VEL
LIN {X 0,Y 262.16,Z 852.793,A -85,B 0,C 180,E1 -13980.029,E2 -13980.029} C_VEL
LIN {X 0,Y 266.8,Z 840.939,A -85,B 0,C 180,E1 -13982.916,E2 -13982.916} C_VEL
LIN {X 0,Y 271.608,Z 827.469,A -85,B 0,C 180,E1 -13985.567,E2 -13985.567} C_VEL
LIN {X 0,Y 276.307,Z 812.619,A -85,B 0,C 180,E1 -13987.919,E2 -13987.919} C_VEL
LIN {X 0,Y 280.522,Z 797.011,A -85,B 0,C 180,E1 -13989.91,E2 -13989.91} C_VEL
LIN {X 0,Y 284.381,Z 779.779,A -85,B 0,C 180,E1 -13991.645,E2 -13991.645} C_VEL
LIN {X 0,Y 287.395,Z 762.516,A -85,B 0,C 180,E1 -13992.993,E2 -13992.993} C_VEL
LIN {X 0,Y 289.658,Z 744.097,A -85,B 0,C 180,E1 -13994.072,E2 -13994.072} C_VEL
LIN {X 0,Y 290.98,Z 725.397,A -85,B 0,C 180,E1 -13994.835,E2 -13994.835} C_VEL
LIN {X 0,Y 293.009,Z 682.119,A -85,B 0,C 180,E1 -13995.959,E2 -13995.959} C_VEL
LIN {X 0,Y 298.034,Z 596.006,A -85,B 0,C 180,E1 -13997.945,E2 -13997.945} C_VEL
LIN {X 0,Y 292.459,Z 604.167,A -85,B 0,C 180,E1 -13998.908,E2 -13998.908} C_VEL
LIN {X 0,Y 288.17,Z 608.506,A -85,B 0,C 180,E1 -13999.763,E2 -13999.763} C_VEL
LIN {X 0,Y 286.304,Z 610.945,A -85,B 0,C 180,E1 -14000.126,E2 -14000.126} C_VEL
LIN {X 0,Y 284.639,Z 615.768,A -85,B 0,C 180,E1 -14000.352,E2 -14000.352} C_VEL
LIN {X 0,Y 282.296,Z 626.6,A -85,B 0,C 180,E1 -14000.513,E2 -14000.513} C_VEL
LIN {X 0,Y 280.461,Z 630.616,A -85,B 0,C 180,E1 -14000.824,E2 -14000.824} C_VEL
LIN {X 0,Y 278.199,Z 633.546,A -85,B 0,C 180,E1 -14001.298,E2 -14001.298} C_VEL
LIN {X 0,Y 272.029,Z 656.403,A -85,B 0,C 180,E1 -14002.016,E2 -14002.016} C_VEL
LIN {X 0,Y 267.137,Z 671.019,A -85,B 0,C 180,E1 -14002.775,E2 -14002.775} C_VEL
LIN {X 0,Y 264.349,Z 676.967,A -85,B 0,C 180,E1 -14003.334,E2 -14003.334} C_VEL
LIN {X 0,Y 263.143,Z 678.144,A -85,B 0,C 180,E1 -14003.647,E2 -14003.647} C_VEL
LIN {X 0,Y 262.785,Z 678.203,A -85,B 0,C 180,E1 -14003.763,E2 -14003.763} C_VEL
LIN {X 0,Y 254.724,Z 753.944,A -85,B 0,C 180,E1 -14007.476,E2 -14007.476} C_VEL
LIN {X 0,Y 252.584,Z 779.808,A -85,B 0,C 180,E1 -14009.028,E2 -14009.028} C_VEL
LIN {X 0,Y 250.669,Z 797.27,A -85,B 0,C 180,E1 -14010.487,E2 -14010.487} C_VEL
LIN {X 0,Y 248.31,Z 814.707,A -85,B 0,C 180,E1 -14012.414,E2 -14012.414} C_VEL
LIN {X 0,Y 245.681,Z 831.336,A -85,B 0,C 180,E1 -14014.786,E2 -14014.786} C_VEL
LIN {X 0,Y 243.183,Z 845.898,A -85,B 0,C 180,E1 -14017.391,E2 -14017.391} C_VEL
LIN {X 0,Y 240.823,Z 859.22,A -85,B 0,C 180,E1 -14020.348,E2 -14020.348} C_VEL
LIN {X 0,Y 238.606,Z 872.19,A -85,B 0,C 180,E1 -14023.944,E2 -14023.944} C_VEL
LIN {X 0,Y 237.03,Z 882.628,A -85,B 0,C 180,E1 -14027.576,E2 -14027.576} C_VEL
LIN {X 0,Y 236.07,Z 891.015,A -85,B 0,C 180,E1 -14031.229,E2 -14031.229} C_VEL
LIN {X 0,Y 235.668,Z 898.745,A -85,B 0,C 180,E1 -14035.619,E2 -14035.619} C_VEL
LIN {X 0,Y 235.985,Z 903.979,A -85,B 0,C 180,E1 -14039.757,E2 -14039.757} C_VEL
LIN {X 0,Y 236.997,Z 907.485,A -85,B 0,C 180,E1 -14043.87,E2 -14043.87} C_VEL
LIN {X 0,Y 238.944,Z 909.358,A -85,B 0,C 180,E1 -14048.179,E2 -14048.179} C_VEL
LIN {X 0,Y 242.315,Z 909.308,A -85,B 0,C 180,E1 -14052.874,E2 -14052.874} C_VEL
LIN {X 0,Y 247.068,Z 907.127,A -85,B 0,C 180,E1 -14057.425,E2 -14057.425} C_VEL
LIN {X 0,Y 253.256,Z 902.86,A -85,B 0,C 180,E1 -14061.784,E2 -14061.784} C_VEL
LIN {X 0,Y 260.516,Z 896.893,A -85,B 0,C 180,E1 -14065.701,E2 -14065.701} C_VEL
LIN {X 0,Y 269.176,Z 889.115,A -85,B 0,C 180,E1 -14069.361,E2 -14069.361} C_VEL
LIN {X 0,Y 279.884,Z 879.056,A -85,B 0,C 180,E1 -14072.888,E2 -14072.888} C_VEL
LIN {X 0,Y 292.367,Z 867.188,A -85,B 0,C 180,E1 -14076.03,E2 -14076.03} C_VEL
LIN {X 0,Y 294.657,Z 865.072,A -85,B 0,C 180,E1 -14076.563,E2 -14076.563} C_VEL
LIN {X 0,Y 279.415,Z 883.618,A -85,B 0,C 180,E1 -14080.098,E2 -14080.098} C_VEL
LIN {X 0,Y 264.339,Z 903.878,A -85,B 0,C 180,E1 -14085.017,E2 -14085.017} C_VEL
LIN {X 0,Y 252.356,Z 922.391,A -85,B 0,C 180,E1 -14090.658,E2 -14090.658} C_VEL
LIN {X 0,Y 244.255,Z 937.093,A -85,B 0,C 180,E1 -14096.198,E2 -14096.198} C_VEL
LIN {X 0,Y 238.782,Z 949.129,A -85,B 0,C 180,E1 -14101.759,E2 -14101.759} C_VEL
LIN {X 0,Y 235.312,Z 959.125,A -85,B 0,C 180,E1 -14107.516,E2 -14107.516} C_VEL
LIN {X 0,Y 233.724,Z 966.339,A -85,B 0,C 180,E1 -14112.831,E2 -14112.831} C_VEL
LIN {X 0,Y 233.306,Z 971.717,A -85,B 0,C 180,E1 -14118.128,E2 -14118.128} C_VEL
LIN {X 0,Y 233.589,Z 974.862,A -85,B 0,C 180,E1 -14122.869,E2 -14122.869} C_VEL
LIN {X 0,Y 233.963,Z 976.225,A -85,B 0,C 180,E1 -14126.815,E2 -14126.815} C_VEL
LIN {X 0,Y 234.132,Z 976.31,A -85,B 0,C 180,E1 -14130.733,E2 -14130.733} C_VEL
LIN {X 0,Y 233.98,Z 975.064,A -85,B 0,C 180,E1 -14134.656,E2 -14134.656} C_VEL
LIN {X 0,Y 233.691,Z 972.28,A -85,B 0,C 180,E1 -14138.86,E2 -14138.86} C_VEL
LIN {X 0,Y 233.665,Z 967.949,A -85,B 0,C 180,E1 -14143.107,E2 -14143.107} C_VEL
LIN {X 0,Y 234.246,Z 961.299,A -85,B 0,C 180,E1 -14147.897,E2 -14147.897} C_VEL
LIN {X 0,Y 235.775,Z 952.582,A -85,B 0,C 180,E1 -14152.699,E2 -14152.699} C_VEL
LIN {X 0,Y 238.408,Z 941.669,A -85,B 0,C 180,E1 -14157.472,E2 -14157.472} C_VEL
LIN {X 0,Y 242.025,Z 929.084,A -85,B 0,C 180,E1 -14161.923,E2 -14161.923} C_VEL
LIN {X 0,Y 246.496,Z 914.928,A -85,B 0,C 180,E1 -14166.026,E2 -14166.026} C_VEL
LIN {X 0,Y 251.813,Z 898.752,A -85,B 0,C 180,E1 -14169.875,E2 -14169.875} C_VEL
LIN {X 0,Y 257.906,Z 880.405,A -85,B 0,C 180,E1 -14173.445,E2 -14173.445} C_VEL
LIN {X 0,Y 264.034,Z 861.208,A -85,B 0,C 180,E1 -14176.483,E2 -14176.483} C_VEL
LIN {X 0,Y 270.613,Z 839.935,A -85,B 0,C 180,E1 -14179.237,E2 -14179.237} C_VEL
LIN {X 0,Y 276.982,Z 817.716,A -85,B 0,C 180,E1 -14181.566,E2 -14181.566} C_VEL
LIN {X 0,Y 282.709,Z 795.864,A -85,B 0,C 180,E1 -14183.401,E2 -14183.401} C_VEL
LIN {X 0,Y 288.065,Z 772.937,A -85,B 0,C 180,E1 -14184.912,E2 -14184.912} C_VEL
LIN {X 0,Y 292.788,Z 748.289,A -85,B 0,C 180,E1 -14186.153,E2 -14186.153} C_VEL
LIN {X 0,Y 296.236,Z 723.571,A -85,B 0,C 180,E1 -14187.076,E2 -14187.076} C_VEL
LIN {X 0,Y 300.652,Z 697.006,A -85,B 0,C 180,E1 -14187.684,E2 -14187.684} C_VEL
LIN {X 0,Y 301.407,Z 694.507,A -85,B 0,C 180,E1 -14187.769,E2 -14187.769} C_VEL
LIN {X 0,Y 315.652,Z 665.144,A -85,B 0,C 180,E1 -14189.316,E2 -14189.316} C_VEL
LIN {X 0,Y 323.003,Z 650.863,A -85,B 0,C 180,E1 -14189.972,E2 -14189.972} C_VEL
LIN {X 0,Y 319.793,Z 630.052,A -85,B 0,C 180,E1 -14193.142,E2 -14193.142} C_VEL
LIN {X 0,Y 318.915,Z 607.811,A -85,B 0,C 180,E1 -14196.272,E2 -14196.272} C_VEL
LIN {X 0,Y 320.493,Z 583.621,A -85,B 0,C 180,E1 -14199.377,E2 -14199.377} C_VEL
LIN {X 0,Y 324.203,Z 559.772,A -85,B 0,C 180,E1 -14202.13,E2 -14202.13} C_VEL
LIN {X 0,Y 316.423,Z 544.165,A -85,B 0,C 180,E1 -14206.292,E2 -14206.292} C_VEL
LIN {X 0,Y 309,Z 529.879,A -85,B 0,C 180,E1 -14210.502,E2 -14210.502} C_VEL
LIN {X 0,Y 301.848,Z 516.545,A -85,B 0,C 180,E1 -14214.869,E2 -14214.869} C_VEL
LIN {X 0,Y 295.606,Z 504.944,A -85,B 0,C 180,E1 -14219.032,E2 -14219.032} C_VEL
LIN {X 0,Y 288.403,Z 492.034,A -85,B 0,C 180,E1 -14224.176,E2 -14224.176} C_VEL
LIN {X 0,Y 283.478,Z 483.577,A -85,B 0,C 180,E1 -14227.907,E2 -14227.907} C_VEL
LIN {X 0,Y 279.141,Z 475.741,A -85,B 0,C 180,E1 -14231.572,E2 -14231.572} C_VEL
LIN {X 0,Y 275.289,Z 469.152,A -85,B 0,C 180,E1 -14234.958,E2 -14234.958} C_VEL
LIN {X 0,Y 273.026,Z 465.158,A -85,B 0,C 180,E1 -14237.097,E2 -14237.097} C_VEL
LIN {X 0,Y 270.426,Z 460.591,A -85,B 0,C 180,E1 -14239.662,E2 -14239.662} C_VEL
LIN {X 0,Y 270.098,Z 460.066,A -85,B 0,C 180,E1 -14240.025,E2 -14240.025} C_VEL
LIN {X 0,Y 275.126,Z 459.335,A -85,B 0,C 180,E1 -14242.658,E2 -14242.658} C_VEL
LIN {X 0,Y 276.62,Z 459.4,A -85,B 0,C 180,E1 -14243.429,E2 -14243.429} C_VEL
LIN {X 0,Y 281.014,Z 467.927,A -85,B 0,C 180,E1 -14246.864,E2 -14246.864} C_VEL
LIN {X 0,Y 286.324,Z 479.4,A -85,B 0,C 180,E1 -14250.654,E2 -14250.654} C_VEL
LIN {X 0,Y 291.78,Z 492.935,A -85,B 0,C 180,E1 -14254.326,E2 -14254.326} C_VEL
LIN {X 0,Y 296.616,Z 506.857,A -85,B 0,C 180,E1 -14257.478,E2 -14257.478} C_VEL
LIN {X 0,Y 297.695,Z 510.423,A -85,B 0,C 180,E1 -14258.194,E2 -14258.194} C_VEL
LIN {X 0,Y 296.712,Z 521.593,A -85,B 0,C 180,E1 -14259.118,E2 -14259.118} C_VEL
LIN {X 0,Y 297.036,Z 528.77,A -85,B 0,C 180,E1 -14259.473,E2 -14259.473} C_VEL
LIN {X 0,Y 285.797,Z 714.41,A -85,B 0,C 180,E1 -14263.794,E2 -14263.794} C_VEL
LIN {X 0,Y 284.682,Z 736.473,A -85,B 0,C 180,E1 -14264.523,E2 -14264.523} C_VEL
LIN {X 0,Y 282.737,Z 755.428,A -85,B 0,C 180,E1 -14265.487,E2 -14265.487} C_VEL
LIN {X 0,Y 279.986,Z 773.021,A -85,B 0,C 180,E1 -14266.714,E2 -14266.714} C_VEL
LIN {X 0,Y 276.385,Z 790.192,A -85,B 0,C 180,E1 -14268.269,E2 -14268.269} C_VEL
LIN {X 0,Y 272.18,Z 806.489,A -85,B 0,C 180,E1 -14270.155,E2 -14270.155} C_VEL
LIN {X 0,Y 267.568,Z 821.573,A -85,B 0,C 180,E1 -14272.341,E2 -14272.341} C_VEL
LIN {X 0,Y 262.562,Z 835.792,A -85,B 0,C 180,E1 -14274.9,E2 -14274.9} C_VEL
LIN {X 0,Y 257.412,Z 848.941,A -85,B 0,C 180,E1 -14277.85,E2 -14277.85} C_VEL
LIN {X 0,Y 252.463,Z 860.546,A -85,B 0,C 180,E1 -14281.108,E2 -14281.108} C_VEL
LIN {X 0,Y 247.868,Z 870.673,A -85,B 0,C 180,E1 -14284.686,E2 -14284.686} C_VEL
LIN {X 0,Y 243.815,Z 879.313,A -85,B 0,C 180,E1 -14288.594,E2 -14288.594} C_VEL
LIN {X 0,Y 240.441,Z 886.441,A -85,B 0,C 180,E1 -14292.828,E2 -14292.828} C_VEL
LIN {X 0,Y 237.989,Z 891.755,A -85,B 0,C 180,E1 -14297.135,E2 -14297.135} C_VEL
LIN {X 0,Y 236.34,Z 895.559,A -85,B 0,C 180,E1 -14301.731,E2 -14301.731} C_VEL
LIN {X 0,Y 235.488,Z 897.665,A -85,B 0,C 180,E1 -14306.349,E2 -14306.349} C_VEL
LIN {X 0,Y 235.305,Z 898.149,A -85,B 0,C 180,E1 -14310.975,E2 -14310.975} C_VEL
LIN {X 0,Y 235.751,Z 897.028,A -85,B 0,C 180,E1 -14315.599,E2 -14315.599} C_VEL
LIN {X 0,Y 236.9,Z 894.259,A -85,B 0,C 180,E1 -14320.211,E2 -14320.211} C_VEL
LIN {X 0,Y 238.924,Z 889.735,A -85,B 0,C 180,E1 -14324.791,E2 -14324.791} C_VEL
LIN {X 0,Y 241.772,Z 883.682,A -85,B 0,C 180,E1 -14329.07,E2 -14329.07} C_VEL
LIN {X 0,Y 245.307,Z 876.21,A -85,B 0,C 180,E1 -14333.036,E2 -14333.036} C_VEL
LIN {X 0,Y 249.415,Z 867.382,A -85,B 0,C 180,E1 -14336.679,E2 -14336.679} C_VEL
LIN {X 0,Y 253.951,Z 857.253,A -85,B 0,C 180,E1 -14340.002,E2 -14340.002} C_VEL
LIN {X 0,Y 258.731,Z 845.848,A -85,B 0,C 180,E1 -14343.018,E2 -14343.018} C_VEL
LIN {X 0,Y 263.823,Z 832.6,A -85,B 0,C 180,E1 -14345.842,E2 -14345.842} C_VEL
LIN {X 0,Y 268.636,Z 818.585,A -85,B 0,C 180,E1 -14348.247,E2 -14348.247} C_VEL
LIN {X 0,Y 273.192,Z 803.219,A -85,B 0,C 180,E1 -14350.377,E2 -14350.377} C_VEL
LIN {X 0,Y 277.179,Z 787.259,A -85,B 0,C 180,E1 -14352.141,E2 -14352.141} C_VEL
LIN {X 0,Y 280.554,Z 770.494,A -85,B 0,C 180,E1 -14353.6,E2 -14353.6} C_VEL
LIN {X 0,Y 283.265,Z 752.235,A -85,B 0,C 180,E1 -14354.817,E2 -14354.817} C_VEL
LIN {X 0,Y 285.053,Z 733.28,A -85,B 0,C 180,E1 -14355.722,E2 -14355.722} C_VEL
LIN {X 0,Y 286.512,Z 701.243,A -85,B 0,C 180,E1 -14356.665,E2 -14356.665} C_VEL
LIN {X 0,Y 291.71,Z 614.009,A -85,B 0,C 180,E1 -14358.714,E2 -14358.714} C_VEL
LIN {X 0,Y 289.068,Z 616.359,A -85,B 0,C 180,E1 -14359.245,E2 -14359.245} C_VEL
LIN {X 0,Y 283.171,Z 626.197,A -85,B 0,C 180,E1 -14360.307,E2 -14360.307} C_VEL
LIN {X 0,Y 280.461,Z 630.616,A -85,B 0,C 180,E1 -14360.824,E2 -14360.824} C_VEL
LIN {X 0,Y 279.139,Z 633.732,A -85,B 0,C 180,E1 -14361.042,E2 -14361.042} C_VEL
LIN {X 0,Y 278.46,Z 638.858,A -85,B 0,C 180,E1 -14361.01,E2 -14361.01} C_VEL
LIN {X 0,Y 278.449,Z 650.539,A -85,B 0,C 180,E1 -14360.535,E2 -14360.535} C_VEL
LIN {X 0,Y 277.753,Z 654.427,A -85,B 0,C 180,E1 -14360.557,E2 -14360.557} C_VEL
LIN {X 0,Y 272.286,Z 671.427,A -85,B 0,C 180,E1 -14361.304,E2 -14361.304} C_VEL
LIN {X 0,Y 268.558,Z 680.179,A -85,B 0,C 180,E1 -14361.962,E2 -14361.962} C_VEL
LIN {X 0,Y 266.119,Z 684.275,A -85,B 0,C 180,E1 -14362.481,E2 -14362.481} C_VEL
LIN {X 0,Y 259.984,Z 706.807,A -85,B 0,C 180,E1 -14363.288,E2 -14363.288} C_VEL
LIN {X 0,Y 254.882,Z 722.203,A -85,B 0,C 180,E1 -14364.162,E2 -14364.162} C_VEL
LIN {X 0,Y 251.877,Z 728.936,A -85,B 0,C 180,E1 -14364.82,E2 -14364.82} C_VEL
LIN {X 0,Y 250.525,Z 730.478,A -85,B 0,C 180,E1 -14365.199,E2 -14365.199} C_VEL
LIN {X 0,Y 250.024,Z 730.474,A -85,B 0,C 180,E1 -14365.38,E2 -14365.38} C_VEL
LIN {X 0,Y 245.811,Z 774.083,A -85,B 0,C 180,E1 -14367.877,E2 -14367.877} C_VEL
LIN {X 0,Y 244.052,Z 791.339,A -85,B 0,C 180,E1 -14369.194,E2 -14369.194} C_VEL
LIN {X 0,Y 241.681,Z 809.39,A -85,B 0,C 180,E1 -14371.05,E2 -14371.05} C_VEL
LIN {X 0,Y 239.201,Z 825.243,A -85,B 0,C 180,E1 -14373.163,E2 -14373.163} C_VEL
LIN {X 0,Y 236.618,Z 840.248,A -85,B 0,C 180,E1 -14375.669,E2 -14375.669} C_VEL
LIN {X 0,Y 233.87,Z 855.338,A -85,B 0,C 180,E1 -14378.822,E2 -14378.822} C_VEL
LIN {X 0,Y 231.577,Z 868.075,A -85,B 0,C 180,E1 -14382.148,E2 -14382.148} C_VEL
LIN {X 0,Y 229.785,Z 878.89,A -85,B 0,C 180,E1 -14385.639,E2 -14385.639} C_VEL
LIN {X 0,Y 228.435,Z 888.863,A -85,B 0,C 180,E1 -14389.661,E2 -14389.661} C_VEL
LIN {X 0,Y 227.794,Z 896.678,A -85,B 0,C 180,E1 -14393.699,E2 -14393.699} C_VEL
LIN {X 0,Y 227.811,Z 902.675,A -85,B 0,C 180,E1 -14397.735,E2 -14397.735} C_VEL
LIN {X 0,Y 228.59,Z 907.444,A -85,B 0,C 180,E1 -14402.255,E2 -14402.255} C_VEL
LIN {X 0,Y 230.138,Z 910.185,A -85,B 0,C 180,E1 -14406.485,E2 -14406.485} C_VEL
LIN {X 0,Y 232.792,Z 911.355,A -85,B 0,C 180,E1 -14410.893,E2 -14410.893} C_VEL
LIN {X 0,Y 237.081,Z 910.601,A -85,B 0,C 180,E1 -14415.658,E2 -14415.658} C_VEL
LIN {X 0,Y 242.845,Z 907.797,A -85,B 0,C 180,E1 -14420.233,E2 -14420.233} C_VEL
LIN {X 0,Y 250.12,Z 903,A -85,B 0,C 180,E1 -14424.565,E2 -14424.565} C_VEL
LIN {X 0,Y 258.498,Z 896.672,A -85,B 0,C 180,E1 -14428.408,E2 -14428.408} C_VEL
LIN {X 0,Y 269.459,Z 887.748,A -85,B 0,C 180,E1 -14432.298,E2 -14432.298} C_VEL
LIN {X 0,Y 282.31,Z 876.938,A -85,B 0,C 180,E1 -14435.759,E2 -14435.759} C_VEL
LIN {X 0,Y 285.186,Z 874.55,A -85,B 0,C 180,E1 -14436.454,E2 -14436.454} C_VEL
LIN {X 0,Y 270.211,Z 891.262,A -85,B 0,C 180,E1 -14440.079,E2 -14440.079} C_VEL
LIN {X 0,Y 255.213,Z 909.88,A -85,B 0,C 180,E1 -14445.162,E2 -14445.162} C_VEL
LIN {X 0,Y 243.276,Z 927.051,A -85,B 0,C 180,E1 -14451.036,E2 -14451.036} C_VEL
LIN {X 0,Y 234.788,Z 941.609,A -85,B 0,C 180,E1 -14457.258,E2 -14457.258} C_VEL
LIN {X 0,Y 229.347,Z 953.374,A -85,B 0,C 180,E1 -14463.596,E2 -14463.596} C_VEL
LIN {X 0,Y 226.586,Z 961.755,A -85,B 0,C 180,E1 -14469.327,E2 -14469.327} C_VEL
LIN {X 0,Y 225.457,Z 967.971,A -85,B 0,C 180,E1 -14474.831,E2 -14474.831} C_VEL
LIN {X 0,Y 225.435,Z 972.046,A -85,B 0,C 180,E1 -14479.935,E2 -14479.935} C_VEL
LIN {X 0,Y 225.883,Z 974.335,A -85,B 0,C 180,E1 -14484.666,E2 -14484.666} C_VEL
LIN {X 0,Y 226.209,Z 974.998,A -85,B 0,C 180,E1 -14488.733,E2 -14488.733} C_VEL
LIN {X 0,Y 226.23,Z 974.405,A -85,B 0,C 180,E1 -14492.532,E2 -14492.532} C_VEL
LIN {X 0,Y 225.965,Z 972.457,A -85,B 0,C 180,E1 -14496.606,E2 -14496.606} C_VEL
LIN {X 0,Y 225.753,Z 968.885,A -85,B 0,C 180,E1 -14500.978,E2 -14500.978} C_VEL
LIN {X 0,Y 226.009,Z 963.048,A -85,B 0,C 180,E1 -14505.919,E2 -14505.919} C_VEL
LIN {X 0,Y 227.042,Z 955.641,A -85,B 0,C 180,E1 -14510.628,E2 -14510.628} C_VEL
LIN {X 0,Y 229.089,Z 946.201,A -85,B 0,C 180,E1 -14515.386,E2 -14515.386} C_VEL
LIN {X 0,Y 232.276,Z 934.599,A -85,B 0,C 180,E1 -14520.093,E2 -14520.093} C_VEL
LIN {X 0,Y 236.477,Z 921.209,A -85,B 0,C 180,E1 -14524.511,E2 -14524.511} C_VEL
LIN {X 0,Y 241.632,Z 905.783,A -85,B 0,C 180,E1 -14528.669,E2 -14528.669} C_VEL
LIN {X 0,Y 247.118,Z 889.705,A -85,B 0,C 180,E1 -14532.233,E2 -14532.233} C_VEL
LIN {X 0,Y 253.348,Z 871.243,A -85,B 0,C 180,E1 -14535.588,E2 -14535.588} C_VEL
LIN {X 0,Y 260.201,Z 850.095,A -85,B 0,C 180,E1 -14538.697,E2 -14538.697} C_VEL
LIN {X 0,Y 266.774,Z 828.708,A -85,B 0,C 180,E1 -14541.252,E2 -14541.252} C_VEL
LIN {X 0,Y 272.94,Z 807.015,A -85,B 0,C 180,E1 -14543.346,E2 -14543.346} C_VEL
LIN {X 0,Y 278.826,Z 783.943,A -85,B 0,C 180,E1 -14545.113,E2 -14545.113} C_VEL
LIN {X 0,Y 284.129,Z 760.122,A -85,B 0,C 180,E1 -14546.512,E2 -14546.512} C_VEL
LIN {X 0,Y 288.26,Z 735.667,A -85,B 0,C 180,E1 -14547.617,E2 -14547.617} C_VEL
LIN {X 0,Y 291.755,Z 711.832,A -85,B 0,C 180,E1 -14548.353,E2 -14548.353} C_VEL
LIN {X 0,Y 295.288,Z 693.911,A -85,B 0,C 180,E1 -14548.756,E2 -14548.756} C_VEL
LIN {X 0,Y 308.755,Z 666.47,A -85,B 0,C 180,E1 -14550.212,E2 -14550.212} C_VEL
LIN {X 0,Y 316.101,Z 652.388,A -85,B 0,C 180,E1 -14550.849,E2 -14550.849} C_VEL
LIN {X 0,Y 313.232,Z 631.379,A -85,B 0,C 180,E1 -14554.068,E2 -14554.068} C_VEL
LIN {X 0,Y 312.71,Z 609.026,A -85,B 0,C 180,E1 -14557.24,E2 -14557.24} C_VEL
LIN {X 0,Y 314.657,Z 584.459,A -85,B 0,C 180,E1 -14560.414,E2 -14560.414} C_VEL
LIN {X 0,Y 317.978,Z 563.734,A -85,B 0,C 180,E1 -14562.856,E2 -14562.856} C_VEL
LIN {X 0,Y 310.682,Z 549.176,A -85,B 0,C 180,E1 -14566.792,E2 -14566.792} C_VEL
LIN {X 0,Y 303.323,Z 534.838,A -85,B 0,C 180,E1 -14571.088,E2 -14571.088} C_VEL
LIN {X 0,Y 295.625,Z 520.287,A -85,B 0,C 180,E1 -14575.928,E2 -14575.928} C_VEL
LIN {X 0,Y 288.443,Z 507.187,A -85,B 0,C 180,E1 -14580.795,E2 -14580.795} C_VEL
LIN {X 0,Y 282.643,Z 496.708,A -85,B 0,C 180,E1 -14585.074,E2 -14585.074} C_VEL
LIN {X 0,Y 276.894,Z 486.542,A -85,B 0,C 180,E1 -14589.671,E2 -14589.671} C_VEL
LIN {X 0,Y 271.936,Z 477.614,A -85,B 0,C 180,E1 -14594.045,E2 -14594.045} C_VEL
LIN {X 0,Y 268.087,Z 471.136,A -85,B 0,C 180,E1 -14597.584,E2 -14597.584} C_VEL
LIN {X 0,Y 266.454,Z 467.844,A -85,B 0,C 180,E1 -14599.396,E2 -14599.396} C_VEL
LIN {X 0,Y 273.599,Z 466.901,A -85,B 0,C 180,E1 -14603.247,E2 -14603.247} C_VEL
LIN {X 0,Y 277.49,Z 475.108,A -85,B 0,C 180,E1 -14606.539,E2 -14606.539} C_VEL
LIN {X 0,Y 282.429,Z 486.04,A -85,B 0,C 180,E1 -14610.18,E2 -14610.18} C_VEL
LIN {X 0,Y 287.549,Z 499.252,A -85,B 0,C 180,E1 -14613.804,E2 -14613.804} C_VEL
LIN {X 0,Y 292.099,Z 512.907,A -85,B 0,C 180,E1 -14616.923,E2 -14616.923} C_VEL
LIN {X 0,Y 292.459,Z 514.69,A -85,B 0,C 180,E1 -14617.239,E2 -14617.239} C_VEL
LIN {X 0,Y 291.761,Z 522.957,A -85,B 0,C 180,E1 -14617.916,E2 -14617.916} C_VEL
LIN {X 0,Y 292.031,Z 530.145,A -85,B 0,C 180,E1 -14618.274,E2 -14618.274} C_VEL
LIN {X 0,Y 280.393,Z 714.879,A -85,B 0,C 180,E1 -14622.604,E2 -14622.604} C_VEL
LIN {X 0,Y 279.223,Z 737.222,A -85,B 0,C 180,E1 -14623.344,E2 -14623.344} C_VEL
LIN {X 0,Y 277.249,Z 755.935,A -85,B 0,C 180,E1 -14624.296,E2 -14624.296} C_VEL
LIN {X 0,Y 274.285,Z 774.261,A -85,B 0,C 180,E1 -14625.582,E2 -14625.582} C_VEL
LIN {X 0,Y 270.539,Z 791.439,A -85,B 0,C 180,E1 -14627.155,E2 -14627.155} C_VEL
LIN {X 0,Y 266.197,Z 807.614,A -85,B 0,C 180,E1 -14629.048,E2 -14629.048} C_VEL
LIN {X 0,Y 261.263,Z 823.107,A -85,B 0,C 180,E1 -14631.327,E2 -14631.327} C_VEL
LIN {X 0,Y 256.017,Z 837.357,A -85,B 0,C 180,E1 -14633.943,E2 -14633.943} C_VEL
LIN {X 0,Y 250.747,Z 850.203,A -85,B 0,C 180,E1 -14636.888,E2 -14636.888} C_VEL
LIN {X 0,Y 245.56,Z 861.811,A -85,B 0,C 180,E1 -14640.215,E2 -14640.215} C_VEL
LIN {X 0,Y 240.73,Z 871.939,A -85,B 0,C 180,E1 -14643.88,E2 -14643.88} C_VEL
LIN {X 0,Y 236.453,Z 880.58,A -85,B 0,C 180,E1 -14647.893,E2 -14647.893} C_VEL
LIN {X 0,Y 232.883,Z 887.708,A -85,B 0,C 180,E1 -14652.253,E2 -14652.253} C_VEL
LIN {X 0,Y 230.276,Z 893.022,A -85,B 0,C 180,E1 -14656.696,E2 -14656.696} C_VEL
LIN {X 0,Y 228.514,Z 896.825,A -85,B 0,C 180,E1 -14661.445,E2 -14661.445} C_VEL
LIN {X 0,Y 227.602,Z 898.929,A -85,B 0,C 180,E1 -14666.222,E2 -14666.222} C_VEL
LIN {X 0,Y 227.406,Z 899.413,A -85,B 0,C 180,E1 -14671.008,E2 -14671.008} C_VEL
LIN {X 0,Y 227.885,Z 898.291,A -85,B 0,C 180,E1 -14675.793,E2 -14675.793} C_VEL
LIN {X 0,Y 229.114,Z 895.524,A -85,B 0,C 180,E1 -14680.562,E2 -14680.562} C_VEL
LIN {X 0,Y 231.273,Z 891,A -85,B 0,C 180,E1 -14685.292,E2 -14685.292} C_VEL
LIN {X 0,Y 234.296,Z 884.947,A -85,B 0,C 180,E1 -14689.703,E2 -14689.703} C_VEL
LIN {X 0,Y 238.033,Z 877.474,A -85,B 0,C 180,E1 -14693.782,E2 -14693.782} C_VEL
LIN {X 0,Y 242.362,Z 868.644,A -85,B 0,C 180,E1 -14697.52,E2 -14697.52} C_VEL
LIN {X 0,Y 247.468,Z 857.781,A -85,B 0,C 180,E1 -14701.143,E2 -14701.143} C_VEL
LIN {X 0,Y 252.898,Z 845.34,A -85,B 0,C 180,E1 -14704.429,E2 -14704.429} C_VEL
LIN {X 0,Y 258.289,Z 831.71,A -85,B 0,C 180,E1 -14707.289,E2 -14707.289} C_VEL
LIN {X 0,Y 263.434,Z 816.974,A -85,B 0,C 180,E1 -14709.758,E2 -14709.758} C_VEL
LIN {X 0,Y 268.135,Z 801.212,A -85,B 0,C 180,E1 -14711.874,E2 -14711.874} C_VEL
LIN {X 0,Y 272.075,Z 785.482,A -85,B 0,C 180,E1 -14713.556,E2 -14713.556} C_VEL
LIN {X 0,Y 275.486,Z 768.343,A -85,B 0,C 180,E1 -14714.993,E2 -14714.993} C_VEL
LIN {X 0,Y 278.091,Z 750.181,A -85,B 0,C 180,E1 -14716.147,E2 -14716.147} C_VEL
LIN {X 0,Y 279.734,Z 731.636,A -85,B 0,C 180,E1 -14716.986,E2 -14716.986} C_VEL
LIN {X 0,Y 281.769,Z 690.876,A -85,B 0,C 180,E1 -14718.129,E2 -14718.129} C_VEL
LIN {X 0,Y 285.312,Z 633.325,A -85,B 0,C 180,E1 -14719.497,E2 -14719.497} C_VEL
LIN {X 0,Y 282.098,Z 638.386,A -85,B 0,C 180,E1 -14720.093,E2 -14720.093} C_VEL
LIN {X 0,Y 277.753,Z 654.427,A -85,B 0,C 180,E1 -14720.557,E2 -14720.557} C_VEL
LIN {X 0,Y 274.252,Z 669.129,A -85,B 0,C 180,E1 -14720.872,E2 -14720.872} C_VEL
LIN {X 0,Y 270.123,Z 688.191,A -85,B 0,C 180,E1 -14721.183,E2 -14721.183} C_VEL
LIN {X 0,Y 263.729,Z 710.978,A -85,B 0,C 180,E1 -14721.986,E2 -14721.986} C_VEL
LIN {X 0,Y 258.47,Z 726.315,A -85,B 0,C 180,E1 -14722.846,E2 -14722.846} C_VEL
LIN {X 0,Y 254.969,Z 733.737,A -85,B 0,C 180,E1 -14723.55,E2 -14723.55} C_VEL
LIN {X 0,Y 252.909,Z 736.887,A -85,B 0,C 180,E1 -14724.023,E2 -14724.023} C_VEL
LIN {X 0,Y 248.058,Z 750.931,A -85,B 0,C 180,E1 -14724.591,E2 -14724.591} C_VEL
LIN {X 0,Y 243.874,Z 759.177,A -85,B 0,C 180,E1 -14725.221,E2 -14725.221} C_VEL
LIN {X 0,Y 241.333,Z 762.544,A -85,B 0,C 180,E1 -14725.776,E2 -14725.776} C_VEL
LIN {X 0,Y 239.703,Z 763.347,A -85,B 0,C 180,E1 -14726.304,E2 -14726.304} C_VEL
LIN {X 0,Y 239.505,Z 763.494,A -85,B 0,C 180,E1 -14726.398,E2 -14726.398} C_VEL
LIN {X 0,Y 237.385,Z 786.001,A -85,B 0,C 180,E1 -14727.946,E2 -14727.946} C_VEL
LIN {X 0,Y 235.017,Z 804.413,A -85,B 0,C 180,E1 -14729.73,E2 -14729.73} C_VEL
LIN {X 0,Y 232.362,Z 821.456,A -85,B 0,C 180,E1 -14731.901,E2 -14731.901} C_VEL
LIN {X 0,Y 229.606,Z 837.299,A -85,B 0,C 180,E1 -14734.461,E2 -14734.461} C_VEL
LIN {X 0,Y 226.853,Z 852.14,A -85,B 0,C 180,E1 -14737.451,E2 -14737.451} C_VEL
LIN {X 0,Y 224.224,Z 866.102,A -85,B 0,C 180,E1 -14741.002,E2 -14741.002} C_VEL
LIN {X 0,Y 222.23,Z 877.484,A -85,B 0,C 180,E1 -14744.605,E2 -14744.605} C_VEL
LIN {X 0,Y 220.766,Z 887.487,A -85,B 0,C 180,E1 -14748.505,E2 -14748.505} C_VEL
LIN {X 0,Y 219.903,Z 896.397,A -85,B 0,C 180,E1 -14752.948,E2 -14752.948} C_VEL
LIN {X 0,Y 219.837,Z 903.178,A -85,B 0,C 180,E1 -14757.392,E2 -14757.392} C_VEL
LIN {X 0,Y 220.534,Z 908.109,A -85,B 0,C 180,E1 -14761.818,E2 -14761.818} C_VEL
LIN {X 0,Y 222.196,Z 911.49,A -85,B 0,C 180,E1 -14766.459,E2 -14766.459} C_VEL
LIN {X 0,Y 225.12,Z 913.059,A -85,B 0,C 180,E1 -14771.269,E2 -14771.269} C_VEL
LIN {X 0,Y 229.121,Z 912.804,A -85,B 0,C 180,E1 -14775.697,E2 -14775.697} C_VEL
LIN {X 0,Y 234.396,Z 910.952,A -85,B 0,C 180,E1 -14779.953,E2 -14779.953} C_VEL
LIN {X 0,Y 241.726,Z 907.056,A -85,B 0,C 180,E1 -14784.433,E2 -14784.433} C_VEL
LIN {X 0,Y 251.156,Z 900.979,A -85,B 0,C 180,E1 -14788.796,E2 -14788.796} C_VEL
LIN {X 0,Y 262.41,Z 893.023,A -85,B 0,C 180,E1 -14792.755,E2 -14792.755} C_VEL
LIN {X 0,Y 275.687,Z 883.15,A -85,B 0,C 180,E1 -14796.331,E2 -14796.331} C_VEL
LIN {X 0,Y 259.859,Z 899.448,A -85,B 0,C 180,E1 -14800.372,E2 -14800.372} C_VEL
LIN {X 0,Y 245.024,Z 916.676,A -85,B 0,C 180,E1 -14805.749,E2 -14805.749} C_VEL
LIN {X 0,Y 232.703,Z 933.471,A -85,B 0,C 180,E1 -14812.4,E2 -14812.4} C_VEL
LIN {X 0,Y 224.631,Z 946.978,A -85,B 0,C 180,E1 -14819.21,E2 -14819.21} C_VEL
LIN {X 0,Y 220.121,Z 956.896,A -85,B 0,C 180,E1 -14825.584,E2 -14825.584} C_VEL
LIN {X 0,Y 217.975,Z 964.134,A -85,B 0,C 180,E1 -14831.547,E2 -14831.547} C_VEL
LIN {X 0,Y 217.406,Z 969.2,A -85,B 0,C 180,E1 -14837.246,E2 -14837.246} C_VEL
LIN {X 0,Y 217.706,Z 972.205,A -85,B 0,C 180,E1 -14842.345,E2 -14842.345} C_VEL
LIN {X 0,Y 218.179,Z 973.422,A -85,B 0,C 180,E1 -14846.584,E2 -14846.584} C_VEL
LIN {X 0,Y 218.409,Z 973.368,A -85,B 0,C 180,E1 -14850.524,E2 -14850.524} C_VEL
LIN {X 0,Y 218.272,Z 972.11,A -85,B 0,C 180,E1 -14854.466,E2 -14854.466} C_VEL
LIN {X 0,Y 217.96,Z 969.415,A -85,B 0,C 180,E1 -14858.706,E2 -14858.706} C_VEL
LIN {X 0,Y 217.906,Z 964.699,A -85,B 0,C 180,E1 -14863.533,E2 -14863.533} C_VEL
LIN {X 0,Y 218.52,Z 958.214,A -85,B 0,C 180,E1 -14868.403,E2 -14868.403} C_VEL
LIN {X 0,Y 220.197,Z 949.33,A -85,B 0,C 180,E1 -14873.552,E2 -14873.552} C_VEL
LIN {X 0,Y 223.104,Z 938.17,A -85,B 0,C 180,E1 -14878.654,E2 -14878.654} C_VEL
LIN {X 0,Y 227.096,Z 925.285,A -85,B 0,C 180,E1 -14883.39,E2 -14883.39} C_VEL
LIN {X 0,Y 232.184,Z 910.227,A -85,B 0,C 180,E1 -14887.876,E2 -14887.876} C_VEL
LIN {X 0,Y 238.025,Z 893.585,A -85,B 0,C 180,E1 -14891.905,E2 -14891.905} C_VEL
LIN {X 0,Y 244.246,Z 875.785,A -85,B 0,C 180,E1 -14895.421,E2 -14895.421} C_VEL
LIN {X 0,Y 250.544,Z 857.164,A -85,B 0,C 180,E1 -14898.425,E2 -14898.425} C_VEL
LIN {X 0,Y 257.036,Z 837.13,A -85,B 0,C 180,E1 -14901.076,E2 -14901.076} C_VEL
LIN {X 0,Y 263.813,Z 814.685,A -85,B 0,C 180,E1 -14903.486,E2 -14903.486} C_VEL
LIN {X 0,Y 270.05,Z 791.972,A -85,B 0,C 180,E1 -14905.422,E2 -14905.422} C_VEL
LIN {X 0,Y 275.583,Z 769.237,A -85,B 0,C 180,E1 -14906.939,E2 -14906.939} C_VEL
LIN {X 0,Y 280.324,Z 745.558,A -85,B 0,C 180,E1 -14908.164,E2 -14908.164} C_VEL
LIN {X 0,Y 283.949,Z 721.54,A -85,B 0,C 180,E1 -14909.089,E2 -14909.089} C_VEL
LIN {X 0,Y 288.804,Z 694.3,A -85,B 0,C 180,E1 -14909.719,E2 -14909.719} C_VEL
LIN {X 0,Y 300.176,Z 671.002,A -85,B 0,C 180,E1 -14910.969,E2 -14910.969} C_VEL
LIN {X 0,Y 309.179,Z 653.427,A -85,B 0,C 180,E1 -14911.827,E2 -14911.827} C_VEL
LIN {X 0,Y 306.685,Z 631.334,A -85,B 0,C 180,E1 -14915.233,E2 -14915.233} C_VEL
LIN {X 0,Y 306.645,Z 608.417,A -85,B 0,C 180,E1 -14918.481,E2 -14918.481} C_VEL
LIN {X 0,Y 309.169,Z 583.329,A -85,B 0,C 180,E1 -14921.718,E2 -14921.718} C_VEL
LIN {X 0,Y 311.753,Z 567.789,A -85,B 0,C 180,E1 -14923.556,E2 -14923.556} C_VEL
LIN {X 0,Y 304.371,Z 552.963,A -85,B 0,C 180,E1 -14927.672,E2 -14927.672} C_VEL
LIN {X 0,Y 296.984,Z 538.537,A -85,B 0,C 180,E1 -14932.066,E2 -14932.066} C_VEL
LIN {X 0,Y 289.826,Z 525.085,A -85,B 0,C 180,E1 -14936.638,E2 -14936.638} C_VEL
LIN {X 0,Y 282.996,Z 512.383,A -85,B 0,C 180,E1 -14941.418,E2 -14941.418} C_VEL
LIN {X 0,Y 276.889,Z 501.463,A -85,B 0,C 180,E1 -14946.012,E2 -14946.012} C_VEL
LIN {X 0,Y 271.254,Z 491.414,A -85,B 0,C 180,E1 -14950.621,E2 -14950.621} C_VEL
LIN {X 0,Y 266.925,Z 483.552,A -85,B 0,C 180,E1 -14954.536,E2 -14954.536} C_VEL
LIN {X 0,Y 263.325,Z 477.387,A -85,B 0,C 180,E1 -14957.913,E2 -14957.913} C_VEL
LIN {X 0,Y 262.627,Z 476.106,A -85,B 0,C 180,E1 -14958.651,E2 -14958.651} C_VEL
LIN {X 0,Y 270.176,Z 474.526,A -85,B 0,C 180,E1 -14962.867,E2 -14962.867} C_VEL
LIN {X 0,Y 270.784,Z 475.033,A -85,B 0,C 180,E1 -14963.272,E2 -14963.272} C_VEL
LIN {X 0,Y 274.367,Z 482.922,A -85,B 0,C 180,E1 -14966.398,E2 -14966.398} C_VEL
LIN {X 0,Y 278.616,Z 492.79,A -85,B 0,C 180,E1 -14969.721,E2 -14969.721} C_VEL
LIN {X 0,Y 283.353,Z 505.529,A -85,B 0,C 180,E1 -14973.25,E2 -14973.25} C_VEL
LIN {X 0,Y 287.399,Z 518.241,A -85,B 0,C 180,E1 -14976.185,E2 -14976.185} C_VEL
LIN {X 0,Y 286.945,Z 524.376,A -85,B 0,C 180,E1 -14976.675,E2 -14976.675} C_VEL
LIN {X 0,Y 287.165,Z 531.391,A -85,B 0,C 180,E1 -14977.03,E2 -14977.03} C_VEL
LIN {X 0,Y 275.114,Z 715.348,A -85,B 0,C 180,E1 -14981.368,E2 -14981.368} C_VEL
LIN {X 0,Y 273.861,Z 738.277,A -85,B 0,C 180,E1 -14982.133,E2 -14982.133} C_VEL
LIN {X 0,Y 271.828,Z 756.856,A -85,B 0,C 180,E1 -14983.084,E2 -14983.084} C_VEL
LIN {X 0,Y 268.94,Z 774.276,A -85,B 0,C 180,E1 -14984.303,E2 -14984.303} C_VEL
LIN {X 0,Y 265.043,Z 791.724,A -85,B 0,C 180,E1 -14985.893,E2 -14985.893} C_VEL
LIN {X 0,Y 260.512,Z 808.09,A -85,B 0,C 180,E1 -14987.806,E2 -14987.806} C_VEL
LIN {X 0,Y 255.462,Z 823.447,A -85,B 0,C 180,E1 -14990.068,E2 -14990.068} C_VEL
LIN {X 0,Y 250.207,Z 837.252,A -85,B 0,C 180,E1 -14992.598,E2 -14992.598} C_VEL
LIN {X 0,Y 244.539,Z 850.584,A -85,B 0,C 180,E1 -14995.651,E2 -14995.651} C_VEL
LIN {X 0,Y 239.059,Z 862.345,A -85,B 0,C 180,E1 -14999.04,E2 -14999.04} C_VEL
LIN {X 0,Y 233.932,Z 872.615,A -85,B 0,C 180,E1 -15002.786,E2 -15002.786} C_VEL
LIN {X 0,Y 229.37,Z 881.4,A -85,B 0,C 180,E1 -15006.902,E2 -15006.902} C_VEL
LIN {X 0,Y 225.537,Z 888.646,A -85,B 0,C 180,E1 -15011.387,E2 -15011.387} C_VEL
LIN {X 0,Y 222.576,Z 894.289,A -85,B 0,C 180,E1 -15016.227,E2 -15016.227} C_VEL
LIN {X 0,Y 220.693,Z 898.09,A -85,B 0,C 180,E1 -15021.14,E2 -15021.14} C_VEL
LIN {X 0,Y 219.717,Z 900.193,A -85,B 0,C 180,E1 -15026.087,E2 -15026.087} C_VEL
LIN {X 0,Y 219.507,Z 900.676,A -85,B 0,C 180,E1 -15031.045,E2 -15031.045} C_VEL
LIN {X 0,Y 220.021,Z 899.555,A -85,B 0,C 180,E1 -15036,E2 -15036} C_VEL
LIN {X 0,Y 221.336,Z 896.789,A -85,B 0,C 180,E1 -15040.938,E2 -15040.938} C_VEL
LIN {X 0,Y 223.64,Z 892.265,A -85,B 0,C 180,E1 -15045.827,E2 -15045.827} C_VEL
LIN {X 0,Y 226.849,Z 886.212,A -85,B 0,C 180,E1 -15050.378,E2 -15050.378} C_VEL
LIN {X 0,Y 230.802,Z 878.737,A -85,B 0,C 180,E1 -15054.576,E2 -15054.576} C_VEL
LIN {X 0,Y 235.435,Z 869.769,A -85,B 0,C 180,E1 -15058.465,E2 -15058.465} C_VEL
LIN {X 0,Y 240.726,Z 859.04,A -85,B 0,C 180,E1 -15062.118,E2 -15062.118} C_VEL
LIN {X 0,Y 246.411,Z 846.596,A -85,B 0,C 180,E1 -15065.469,E2 -15065.469} C_VEL
LIN {X 0,Y 252.08,Z 832.863,A -85,B 0,C 180,E1 -15068.396,E2 -15068.396} C_VEL
LIN {X 0,Y 257.414,Z 818.197,A -85,B 0,C 180,E1 -15070.887,E2 -15070.887} C_VEL
LIN {X 0,Y 262.303,Z 802.451,A -85,B 0,C 180,E1 -15073.026,E2 -15073.026} C_VEL
LIN {X 0,Y 266.402,Z 786.713,A -85,B 0,C 180,E1 -15074.727,E2 -15074.727} C_VEL
LIN {X 0,Y 269.871,Z 770.042,A -85,B 0,C 180,E1 -15076.145,E2 -15076.145} C_VEL
LIN {X 0,Y 272.631,Z 751.683,A -85,B 0,C 180,E1 -15077.331,E2 -15077.331} C_VEL
LIN {X 0,Y 274.373,Z 733.005,A -85,B 0,C 180,E1 -15078.188,E2 -15078.188} C_VEL
LIN {X 0,Y 276.495,Z 692.378,A -85,B 0,C 180,E1 -15079.347,E2 -15079.347} C_VEL
LIN {X 0,Y 277.864,Z 670.876,A -85,B 0,C 180,E1 -15079.863,E2 -15079.863} C_VEL
LIN {X 0,Y 273.377,Z 682.215,A -85,B 0,C 180,E1 -15080.561,E2 -15080.561} C_VEL
LIN {X 0,Y 270.123,Z 688.191,A -85,B 0,C 180,E1 -15081.183,E2 -15081.183} C_VEL
LIN {X 0,Y 268.736,Z 695.846,A -85,B 0,C 180,E1 -15081.237,E2 -15081.237} C_VEL
LIN {X 0,Y 266.938,Z 714.658,A -85,B 0,C 180,E1 -15080.925,E2 -15080.925} C_VEL
LIN {X 0,Y 265.268,Z 722.117,A -85,B 0,C 180,E1 -15081.064,E2 -15081.064} C_VEL
LIN {X 0,Y 264.927,Z 723.134,A -85,B 0,C 180,E1 -15081.115,E2 -15081.115} C_VEL
LIN {X 0,Y 260.375,Z 734.307,A -85,B 0,C 180,E1 -15081.863,E2 -15081.863} C_VEL
LIN {X 0,Y 256.722,Z 740.569,A -85,B 0,C 180,E1 -15082.585,E2 -15082.585} C_VEL
LIN {X 0,Y 250.986,Z 755.209,A -85,B 0,C 180,E1 -15083.161,E2 -15083.161} C_VEL
LIN {X 0,Y 246.411,Z 763.587,A -85,B 0,C 180,E1 -15083.778,E2 -15083.778} C_VEL
LIN {X 0,Y 242.915,Z 768.123,A -85,B 0,C 180,E1 -15084.45,E2 -15084.45} C_VEL
LIN {X 0,Y 241.086,Z 769.93,A -85,B 0,C 180,E1 -15084.886,E2 -15084.886} C_VEL
LIN {X 0,Y 237.111,Z 777.073,A -85,B 0,C 180,E1 -15085.3,E2 -15085.3} C_VEL
LIN {X 0,Y 234.44,Z 780.797,A -85,B 0,C 180,E1 -15085.738,E2 -15085.738} C_VEL
LIN {X 0,Y 232.21,Z 782.939,A -85,B 0,C 180,E1 -15086.257,E2 -15086.257} C_VEL
LIN {X 0,Y 230.5,Z 783.573,A -85,B 0,C 180,E1 -15086.868,E2 -15086.868} C_VEL
LIN {X 0,Y 230.344,Z 783.768,A -85,B 0,C 180,E1 -15086.954,E2 -15086.954} C_VEL
LIN {X 0,Y 228.155,Z 800.97,A -85,B 0,C 180,E1 -15088.566,E2 -15088.566} C_VEL
LIN {X 0,Y 225.369,Z 818.983,A -85,B 0,C 180,E1 -15090.789,E2 -15090.789} C_VEL
LIN {X 0,Y 222.369,Z 835.832,A -85,B 0,C 180,E1 -15093.483,E2 -15093.483} C_VEL
LIN {X 0,Y 219.543,Z 850.497,A -85,B 0,C 180,E1 -15096.447,E2 -15096.447} C_VEL
LIN {X 0,Y 216.947,Z 863.868,A -85,B 0,C 180,E1 -15099.777,E2 -15099.777} C_VEL
LIN {X 0,Y 214.604,Z 876.735,A -85,B 0,C 180,E1 -15103.766,E2 -15103.766} C_VEL
LIN {X 0,Y 212.897,Z 887.668,A -85,B 0,C 180,E1 -15108.073,E2 -15108.073} C_VEL
LIN {X 0,Y 211.995,Z 896.408,A -85,B 0,C 180,E1 -15112.411,E2 -15112.411} C_VEL
LIN {X 0,Y 211.847,Z 903.246,A -85,B 0,C 180,E1 -15116.752,E2 -15116.752} C_VEL
LIN {X 0,Y 212.539,Z 908.903,A -85,B 0,C 180,E1 -15121.617,E2 -15121.617} C_VEL
LIN {X 0,Y 214.11,Z 912.497,A -85,B 0,C 180,E1 -15126.165,E2 -15126.165} C_VEL
LIN {X 0,Y 217.071,Z 914.649,A -85,B 0,C 180,E1 -15131.154,E2 -15131.154} C_VEL
LIN {X 0,Y 221.691,Z 914.87,A -85,B 0,C 180,E1 -15136.237,E2 -15136.237} C_VEL
LIN {X 0,Y 228.291,Z 912.984,A -85,B 0,C 180,E1 -15141.316,E2 -15141.316} C_VEL
LIN {X 0,Y 236.235,Z 909.306,A -85,B 0,C 180,E1 -15145.845,E2 -15145.845} C_VEL
LIN {X 0,Y 246.364,Z 903.583,A -85,B 0,C 180,E1 -15150.214,E2 -15150.214} C_VEL
LIN {X 0,Y 258.949,Z 895.694,A -85,B 0,C 180,E1 -15154.314,E2 -15154.314} C_VEL
LIN {X 0,Y 266.035,Z 891.071,A -85,B 0,C 180,E1 -15156.215,E2 -15156.215} C_VEL
LIN {X 0,Y 248.657,Z 907.672,A -85,B 0,C 180,E1 -15160.951,E2 -15160.951} C_VEL
LIN {X 0,Y 233.279,Z 924.582,A -85,B 0,C 180,E1 -15167.131,E2 -15167.131} C_VEL
LIN {X 0,Y 221.565,Z 940.028,A -85,B 0,C 180,E1 -15174.398,E2 -15174.398} C_VEL
LIN {X 0,Y 214.473,Z 951.888,A -85,B 0,C 180,E1 -15181.606,E2 -15181.606} C_VEL
LIN {X 0,Y 210.987,Z 960.056,A -85,B 0,C 180,E1 -15188.013,E2 -15188.013} C_VEL
LIN {X 0,Y 209.581,Z 966.065,A -85,B 0,C 180,E1 -15194.22,E2 -15194.22} C_VEL
LIN {X 0,Y 209.568,Z 969.787,A -85,B 0,C 180,E1 -15199.832,E2 -15199.832} C_VEL
LIN {X 0,Y 210.119,Z 971.652,A -85,B 0,C 180,E1 -15204.812,E2 -15204.812} C_VEL
LIN {X 0,Y 210.503,Z 971.989,A -85,B 0,C 180,E1 -15208.911,E2 -15208.911} C_VEL
LIN {X 0,Y 210.517,Z 971.123,A -85,B 0,C 180,E1 -15212.994,E2 -15212.994} C_VEL
LIN {X 0,Y 210.207,Z 968.8,A -85,B 0,C 180,E1 -15217.378,E2 -15217.378} C_VEL
LIN {X 0,Y 210.002,Z 964.807,A -85,B 0,C 180,E1 -15222.092,E2 -15222.092} C_VEL
LIN {X 0,Y 210.402,Z 958.667,A -85,B 0,C 180,E1 -15227.222,E2 -15227.222} C_VEL
LIN {X 0,Y 211.895,Z 950.031,A -85,B 0,C 180,E1 -15232.763,E2 -15232.763} C_VEL
LIN {X 0,Y 214.285,Z 940.751,A -85,B 0,C 180,E1 -15237.56,E2 -15237.56} C_VEL
LIN {X 0,Y 217.508,Z 930.237,A -85,B 0,C 180,E1 -15241.913,E2 -15241.913} C_VEL
LIN {X 0,Y 221.817,Z 917.358,A -85,B 0,C 180,E1 -15246.211,E2 -15246.211} C_VEL
LIN {X 0,Y 228.782,Z 897.54,A -85,B 0,C 180,E1 -15251.46,E2 -15251.46} C_VEL
LIN {X 0,Y 235.165,Z 879.937,A -85,B 0,C 180,E1 -15255.237,E2 -15255.237} C_VEL
LIN {X 0,Y 241.434,Z 862.043,A -85,B 0,C 180,E1 -15258.374,E2 -15258.374} C_VEL
LIN {X 0,Y 248.447,Z 841.45,A -85,B 0,C 180,E1 -15261.327,E2 -15261.327} C_VEL
LIN {X 0,Y 255.509,Z 819.108,A -85,B 0,C 180,E1 -15263.908,E2 -15263.908} C_VEL
LIN {X 0,Y 262.213,Z 795.853,A -85,B 0,C 180,E1 -15266.032,E2 -15266.032} C_VEL
LIN {X 0,Y 268.234,Z 772.386,A -85,B 0,C 180,E1 -15267.695,E2 -15267.695} C_VEL
LIN {X 0,Y 273.24,Z 748.973,A -85,B 0,C 180,E1 -15268.975,E2 -15268.975} C_VEL
LIN {X 0,Y 277.073,Z 725.136,A -85,B 0,C 180,E1 -15269.979,E2 -15269.979} C_VEL
LIN {X 0,Y 281.948,Z 697.747,A -85,B 0,C 180,E1 -15270.696,E2 -15270.696} C_VEL
LIN {X 0,Y 283.379,Z 691.997,A -85,B 0,C 180,E1 -15270.839,E2 -15270.839} C_VEL
LIN {X 0,Y 295.719,Z 667.636,A -85,B 0,C 180,E1 -15272.147,E2 -15272.147} C_VEL
LIN {X 0,Y 302.377,Z 654.774,A -85,B 0,C 180,E1 -15272.771,E2 -15272.771} C_VEL
LIN {X 0,Y 300.217,Z 631.834,A -85,B 0,C 180,E1 -15276.329,E2 -15276.329} C_VEL
LIN {X 0,Y 300.644,Z 608.171,A -85,B 0,C 180,E1 -15279.693,E2 -15279.693} C_VEL
LIN {X 0,Y 303.631,Z 582.813,A -85,B 0,C 180,E1 -15282.958,E2 -15282.958} C_VEL
LIN {X 0,Y 305.624,Z 572.003,A -85,B 0,C 180,E1 -15284.245,E2 -15284.245} C_VEL
LIN {X 0,Y 298.287,Z 557.22,A -85,B 0,C 180,E1 -15288.398,E2 -15288.398} C_VEL
LIN {X 0,Y 290.911,Z 542.823,A -85,B 0,C 180,E1 -15292.893,E2 -15292.893} C_VEL
LIN {X 0,Y 284.076,Z 529.878,A -85,B 0,C 180,E1 -15297.378,E2 -15297.378} C_VEL
LIN {X 0,Y 277.766,Z 518.093,A -85,B 0,C 180,E1 -15301.857,E2 -15301.857} C_VEL
LIN {X 0,Y 271.702,Z 507.169,A -85,B 0,C 180,E1 -15306.492,E2 -15306.492} C_VEL
LIN {X 0,Y 266.035,Z 496.913,A -85,B 0,C 180,E1 -15311.271,E2 -15311.271} C_VEL
LIN {X 0,Y 261.35,Z 488.572,A -85,B 0,C 180,E1 -15315.534,E2 -15315.534} C_VEL
LIN {X 0,Y 259.069,Z 484.245,A -85,B 0,C 180,E1 -15317.985,E2 -15317.985} C_VEL
LIN {X 0,Y 264.099,Z 482.914,A -85,B 0,C 180,E1 -15321.08,E2 -15321.08} C_VEL
LIN {X 0,Y 267.501,Z 482.18,A -85,B 0,C 180,E1 -15322.876,E2 -15322.876} C_VEL
LIN {X 0,Y 270.978,Z 490.109,A -85,B 0,C 180,E1 -15326.046,E2 -15326.046} C_VEL
LIN {X 0,Y 274.745,Z 499.333,A -85,B 0,C 180,E1 -15329.187,E2 -15329.187} C_VEL
LIN {X 0,Y 279.28,Z 512.018,A -85,B 0,C 180,E1 -15332.725,E2 -15332.725} C_VEL
LIN {X 0,Y 282.413,Z 522.303,A -85,B 0,C 180,E1 -15335.132,E2 -15335.132} C_VEL
LIN {X 0,Y 282.337,Z 527.107,A -85,B 0,C 180,E1 -15335.471,E2 -15335.471} C_VEL
LIN {X 0,Y 282.428,Z 532.802,A -85,B 0,C 180,E1 -15335.748,E2 -15335.748} C_VEL
LIN {X 0,Y 269.972,Z 715.752,A -85,B 0,C 180,E1 -15340.082,E2 -15340.082} C_VEL
LIN {X 0,Y 268.64,Z 739.179,A -85,B 0,C 180,E1 -15340.866,E2 -15340.866} C_VEL
LIN {X 0,Y 266.548,Z 757.674,A -85,B 0,C 180,E1 -15341.816,E2 -15341.816} C_VEL
LIN {X 0,Y 263.574,Z 775.06,A -85,B 0,C 180,E1 -15343.035,E2 -15343.035} C_VEL
LIN {X 0,Y 259.681,Z 792.01,A -85,B 0,C 180,E1 -15344.577,E2 -15344.577} C_VEL
LIN {X 0,Y 254.941,Z 808.62,A -85,B 0,C 180,E1 -15346.516,E2 -15346.516} C_VEL
LIN {X 0,Y 249.472,Z 824.651,A -85,B 0,C 180,E1 -15348.894,E2 -15348.894} C_VEL
LIN {X 0,Y 243.748,Z 839.055,A -85,B 0,C 180,E1 -15351.582,E2 -15351.582} C_VEL
LIN {X 0,Y 238.048,Z 851.846,A -85,B 0,C 180,E1 -15354.576,E2 -15354.576} C_VEL
LIN {X 0,Y 232.305,Z 863.609,A -85,B 0,C 180,E1 -15358.036,E2 -15358.036} C_VEL
LIN {X 0,Y 226.915,Z 873.881,A -85,B 0,C 180,E1 -15361.871,E2 -15361.871} C_VEL
LIN {X 0,Y 222.103,Z 882.667,A -85,B 0,C 180,E1 -15366.1,E2 -15366.1} C_VEL
LIN {X 0,Y 218.042,Z 889.914,A -85,B 0,C 180,E1 -15370.722,E2 -15370.722} C_VEL
LIN {X 0,Y 215.031,Z 895.321,A -85,B 0,C 180,E1 -15375.459,E2 -15375.459} C_VEL
LIN {X 0,Y 212.963,Z 899.21,A -85,B 0,C 180,E1 -15380.543,E2 -15380.543} C_VEL
LIN {X 0,Y 211.869,Z 901.395,A -85,B 0,C 180,E1 -15385.67,E2 -15385.67} C_VEL
LIN {X 0,Y 211.603,Z 901.96,A -85,B 0,C 180,E1 -15390.813,E2 -15390.813} C_VEL
LIN {X 0,Y 212.11,Z 900.923,A -85,B 0,C 180,E1 -15395.953,E2 -15395.953} C_VEL
LIN {X 0,Y 213.47,Z 898.244,A -85,B 0,C 180,E1 -15401.073,E2 -15401.073} C_VEL
LIN {X 0,Y 215.869,Z 893.811,A -85,B 0,C 180,E1 -15406.136,E2 -15406.136} C_VEL
LIN {X 0,Y 219.218,Z 887.855,A -85,B 0,C 180,E1 -15410.841,E2 -15410.841} C_VEL
LIN {X 0,Y 223.618,Z 880.001,A -85,B 0,C 180,E1 -15415.42,E2 -15415.42} C_VEL
LIN {X 0,Y 228.639,Z 870.782,A -85,B 0,C 180,E1 -15419.511,E2 -15419.511} C_VEL
LIN {X 0,Y 234.057,Z 860.299,A -85,B 0,C 180,E1 -15423.148,E2 -15423.148} C_VEL
LIN {X 0,Y 240.011,Z 847.851,A -85,B 0,C 180,E1 -15426.565,E2 -15426.565} C_VEL
LIN {X 0,Y 245.893,Z 834.212,A -85,B 0,C 180,E1 -15429.522,E2 -15429.522} C_VEL
LIN {X 0,Y 251.484,Z 819.465,A -85,B 0,C 180,E1 -15432.063,E2 -15432.063} C_VEL
LIN {X 0,Y 256.582,Z 803.69,A -85,B 0,C 180,E1 -15434.231,E2 -15434.231} C_VEL
LIN {X 0,Y 260.846,Z 787.943,A -85,B 0,C 180,E1 -15435.949,E2 -15435.949} C_VEL
LIN {X 0,Y 264.574,Z 770.561,A -85,B 0,C 180,E1 -15437.431,E2 -15437.431} C_VEL
LIN {X 0,Y 267.395,Z 752.323,A -85,B 0,C 180,E1 -15438.608,E2 -15438.608} C_VEL
LIN {X 0,Y 269.185,Z 733.601,A -85,B 0,C 180,E1 -15439.466,E2 -15439.466} C_VEL
LIN {X 0,Y 270.595,Z 705.324,A -85,B 0,C 180,E1 -15440.335,E2 -15440.335} C_VEL
LIN {X 0,Y 264.927,Z 723.134,A -85,B 0,C 180,E1 -15441.115,E2 -15441.115} C_VEL
LIN {X 0,Y 263.08,Z 730.326,A -85,B 0,C 180,E1 -15441.305,E2 -15441.305} C_VEL
LIN {X 0,Y 260.236,Z 744.369,A -85,B 0,C 180,E1 -15441.244,E2 -15441.244} C_VEL
LIN {X 0,Y 259.544,Z 746.509,A -85,B 0,C 180,E1 -15441.285,E2 -15441.285} C_VEL
LIN {X 0,Y 254.007,Z 759.438,A -85,B 0,C 180,E1 -15441.757,E2 -15441.757} C_VEL
LIN {X 0,Y 248.916,Z 768.131,A -85,B 0,C 180,E1 -15442.369,E2 -15442.369} C_VEL
LIN {X 0,Y 244.654,Z 773.376,A -85,B 0,C 180,E1 -15443.075,E2 -15443.075} C_VEL
LIN {X 0,Y 243.051,Z 775.146,A -85,B 0,C 180,E1 -15443.38,E2 -15443.38} C_VEL
LIN {X 0,Y 238.29,Z 782.708,A -85,B 0,C 180,E1 -15443.875,E2 -15443.875} C_VEL
LIN {X 0,Y 234.385,Z 787.348,A -85,B 0,C 180,E1 -15444.537,E2 -15444.537} C_VEL
LIN {X 0,Y 230.731,Z 790.311,A -85,B 0,C 180,E1 -15445.41,E2 -15445.41} C_VEL
LIN {X 0,Y 226.353,Z 795.957,A -85,B 0,C 180,E1 -15446.027,E2 -15446.027} C_VEL
LIN {X 0,Y 223.631,Z 798.559,A -85,B 0,C 180,E1 -15446.637,E2 -15446.637} C_VEL
LIN {X 0,Y 221.757,Z 799.596,A -85,B 0,C 180,E1 -15447.244,E2 -15447.244} C_VEL
LIN {X 0,Y 221.043,Z 799.636,A -85,B 0,C 180,E1 -15447.586,E2 -15447.586} C_VEL
LIN {X 0,Y 218.438,Z 816.202,A -85,B 0,C 180,E1 -15449.615,E2 -15449.615} C_VEL
LIN {X 0,Y 215.448,Z 832.736,A -85,B 0,C 180,E1 -15452.198,E2 -15452.198} C_VEL
LIN {X 0,Y 212.185,Z 849.357,A -85,B 0,C 180,E1 -15455.5,E2 -15455.5} C_VEL
LIN {X 0,Y 209.269,Z 863.854,A -85,B 0,C 180,E1 -15459.147,E2 -15459.147} C_VEL
LIN {X 0,Y 207.002,Z 875.689,A -85,B 0,C 180,E1 -15462.863,E2 -15462.863} C_VEL
LIN {X 0,Y 205.218,Z 886.55,A -85,B 0,C 180,E1 -15467.048,E2 -15467.048} C_VEL
LIN {X 0,Y 204.117,Z 896.066,A -85,B 0,C 180,E1 -15471.691,E2 -15471.691} C_VEL
LIN {X 0,Y 203.87,Z 903.504,A -85,B 0,C 180,E1 -15476.344,E2 -15476.344} C_VEL
LIN {X 0,Y 204.477,Z 909.321,A -85,B 0,C 180,E1 -15481.12,E2 -15481.12} C_VEL
LIN {X 0,Y 206.26,Z 913.773,A -85,B 0,C 180,E1 -15486.401,E2 -15486.401} C_VEL
LIN {X 0,Y 209.382,Z 916.228,A -85,B 0,C 180,E1 -15491.569,E2 -15491.569} C_VEL
LIN {X 0,Y 213.69,Z 916.857,A -85,B 0,C 180,E1 -15496.304,E2 -15496.304} C_VEL
LIN {X 0,Y 219.745,Z 915.855,A -85,B 0,C 180,E1 -15501.066,E2 -15501.066} C_VEL
LIN {X 0,Y 228.187,Z 912.852,A -85,B 0,C 180,E1 -15505.987,E2 -15505.987} C_VEL
LIN {X 0,Y 238.493,Z 907.991,A -85,B 0,C 180,E1 -15510.482,E2 -15510.482} C_VEL
LIN {X 0,Y 250.65,Z 901.435,A -85,B 0,C 180,E1 -15514.502,E2 -15514.502} C_VEL
LIN {X 0,Y 256.443,Z 898.182,A -85,B 0,C 180,E1 -15516.067,E2 -15516.067} C_VEL
LIN {X 0,Y 238.261,Z 914.265,A -85,B 0,C 180,E1 -15521.307,E2 -15521.307} C_VEL
LIN {X 0,Y 222.347,Z 930.699,A -85,B 0,C 180,E1 -15528.285,E2 -15528.285} C_VEL
LIN {X 0,Y 211.574,Z 944.264,A -85,B 0,C 180,E1 -15535.779,E2 -15535.779} C_VEL
LIN {X 0,Y 205.529,Z 954.125,A -85,B 0,C 180,E1 -15542.787,E2 -15542.787} C_VEL
LIN {X 0,Y 202.39,Z 961.7,A -85,B 0,C 180,E1 -15549.823,E2 -15549.823} C_VEL
LIN {X 0,Y 201.516,Z 966.458,A -85,B 0,C 180,E1 -15555.928,E2 -15555.928} C_VEL
LIN {X 0,Y 201.79,Z 969.282,A -85,B 0,C 180,E1 -15561.451,E2 -15561.451} C_VEL
LIN {X 0,Y 202.415,Z 970.427,A -85,B 0,C 180,E1 -15566.317,E2 -15566.317} C_VEL
LIN {X 0,Y 202.727,Z 970.187,A -85,B 0,C 180,E1 -15570.564,E2 -15570.564} C_VEL
LIN {X 0,Y 202.575,Z 968.685,A -85,B 0,C 180,E1 -15574.812,E2 -15574.812} C_VEL
LIN {X 0,Y 202.211,Z 965.445,A -85,B 0,C 180,E1 -15579.678,E2 -15579.678} C_VEL
LIN {X 0,Y 202.283,Z 959.473,A -85,B 0,C 180,E1 -15585.774,E2 -15585.774} C_VEL
LIN {X 0,Y 203.28,Z 952.796,A -85,B 0,C 180,E1 -15591.042,E2 -15591.042} C_VEL
LIN {X 0,Y 205.445,Z 944.071,A -85,B 0,C 180,E1 -15596.287,E2 -15596.287} C_VEL
LIN {X 0,Y 208.698,Z 933.766,A -85,B 0,C 180,E1 -15601.159,E2 -15601.159} C_VEL
LIN {X 0,Y 212.927,Z 921.787,A -85,B 0,C 180,E1 -15605.673,E2 -15605.673} C_VEL
LIN {X 0,Y 217.935,Z 908.119,A -85,B 0,C 180,E1 -15609.792,E2 -15609.792} C_VEL
LIN {X 0,Y 223.202,Z 893.34,A -85,B 0,C 180,E1 -15613.368,E2 -15613.368} C_VEL
LIN {X 0,Y 228.521,Z 877.655,A -85,B 0,C 180,E1 -15616.395,E2 -15616.395} C_VEL
LIN {X 0,Y 237.704,Z 851.497,A -85,B 0,C 180,E1 -15620.71,E2 -15620.71} C_VEL
LIN {X 0,Y 245.213,Z 829.231,A -85,B 0,C 180,E1 -15623.639,E2 -15623.639} C_VEL
LIN {X 0,Y 252.378,Z 806.214,A -85,B 0,C 180,E1 -15626.041,E2 -15626.041} C_VEL
LIN {X 0,Y 259.06,Z 782.234,A -85,B 0,C 180,E1 -15628.001,E2 -15628.001} C_VEL
LIN {X 0,Y 265.053,Z 757.511,A -85,B 0,C 180,E1 -15629.537,E2 -15629.537} C_VEL
LIN {X 0,Y 269.568,Z 733.036,A -85,B 0,C 180,E1 -15630.717,E2 -15630.717} C_VEL
LIN {X 0,Y 273.679,Z 708.438,A -85,B 0,C 180,E1 -15631.505,E2 -15631.505} C_VEL
LIN {X 0,Y 277.169,Z 691.677,A -85,B 0,C 180,E1 -15631.885,E2 -15631.885} C_VEL
LIN {X 0,Y 289.579,Z 667.414,A -85,B 0,C 180,E1 -15633.194,E2 -15633.194} C_VEL
LIN {X 0,Y 295.575,Z 655.87,A -85,B 0,C 180,E1 -15633.769,E2 -15633.769} C_VEL
LIN {X 0,Y 293.817,Z 632.729,A -85,B 0,C 180,E1 -15637.385,E2 -15637.385} C_VEL
LIN {X 0,Y 294.611,Z 608.968,A -85,B 0,C 180,E1 -15640.78,E2 -15640.78} C_VEL
LIN {X 0,Y 298.06,Z 583.073,A -85,B 0,C 180,E1 -15644.134,E2 -15644.134} C_VEL
LIN {X 0,Y 299.357,Z 576,A -85,B 0,C 180,E1 -15644.989,E2 -15644.989} C_VEL
LIN {X 0,Y 292.139,Z 561.414,A -85,B 0,C 180,E1 -15649.192,E2 -15649.192} C_VEL
LIN {X 0,Y 285.409,Z 548.179,A -85,B 0,C 180,E1 -15653.362,E2 -15653.362} C_VEL
LIN {X 0,Y 278.281,Z 534.551,A -85,B 0,C 180,E1 -15658.147,E2 -15658.147} C_VEL
LIN {X 0,Y 272.23,Z 523.245,A -85,B 0,C 180,E1 -15662.554,E2 -15662.554} C_VEL
LIN {X 0,Y 266.375,Z 512.585,A -85,B 0,C 180,E1 -15667.116,E2 -15667.116} C_VEL
LIN {X 0,Y 260.52,Z 501.801,A -85,B 0,C 180,E1 -15672.187,E2 -15672.187} C_VEL
LIN {X 0,Y 255.735,Z 493.276,A -85,B 0,C 180,E1 -15676.689,E2 -15676.689} C_VEL
LIN {X 0,Y 255.4,Z 492.404,A -85,B 0,C 180,E1 -15677.188,E2 -15677.188} C_VEL
LIN {X 0,Y 261.877,Z 490.554,A -85,B 0,C 180,E1 -15681.268,E2 -15681.268} C_VEL
LIN {X 0,Y 264.776,Z 490.219,A -85,B 0,C 180,E1 -15682.89,E2 -15682.89} C_VEL
LIN {X 0,Y 268.584,Z 499.61,A -85,B 0,C 180,E1 -15686.534,E2 -15686.534} C_VEL
LIN {X 0,Y 272.277,Z 509.564,A -85,B 0,C 180,E1 -15689.72,E2 -15689.72} C_VEL
LIN {X 0,Y 276.141,Z 521.407,A -85,B 0,C 180,E1 -15692.897,E2 -15692.897} C_VEL
LIN {X 0,Y 277.705,Z 526.505,A -85,B 0,C 180,E1 -15694.024,E2 -15694.024} C_VEL
LIN {X 0,Y 277.869,Z 533.776,A -85,B 0,C 180,E1 -15694.413,E2 -15694.413} C_VEL
LIN {X 0,Y 264.961,Z 716.331,A -85,B 0,C 180,E1 -15698.752,E2 -15698.752} C_VEL
LIN {X 0,Y 263.541,Z 740.232,A -85,B 0,C 180,E1 -15699.557,E2 -15699.557} C_VEL
LIN {X 0,Y 261.357,Z 758.799,A -85,B 0,C 180,E1 -15700.517,E2 -15700.517} C_VEL
LIN {X 0,Y 258.23,Z 776.365,A -85,B 0,C 180,E1 -15701.758,E2 -15701.758} C_VEL
LIN {X 0,Y 254.197,Z 793.257,A -85,B 0,C 180,E1 -15703.309,E2 -15703.309} C_VEL
LIN {X 0,Y 249.285,Z 809.818,A -85,B 0,C 180,E1 -15705.259,E2 -15705.259} C_VEL
LIN {X 0,Y 243.754,Z 825.43,A -85,B 0,C 180,E1 -15707.592,E2 -15707.592} C_VEL
LIN {X 0,Y 237.788,Z 839.89,A -85,B 0,C 180,E1 -15710.309,E2 -15710.309} C_VEL
LIN {X 0,Y 231.646,Z 853.109,A -85,B 0,C 180,E1 -15713.442,E2 -15713.442} C_VEL
LIN {X 0,Y 225.627,Z 864.874,A -85,B 0,C 180,E1 -15716.971,E2 -15716.971} C_VEL
LIN {X 0,Y 219.961,Z 875.147,A -85,B 0,C 180,E1 -15720.898,E2 -15720.898} C_VEL
LIN {X 0,Y 214.881,Z 883.934,A -85,B 0,C 180,E1 -15725.243,E2 -15725.243} C_VEL
LIN {X 0,Y 210.578,Z 891.181,A -85,B 0,C 180,E1 -15730.01,E2 -15730.01} C_VEL
LIN {X 0,Y 207.226,Z 896.822,A -85,B 0,C 180,E1 -15735.184,E2 -15735.184} C_VEL
LIN {X 0,Y 205.073,Z 900.621,A -85,B 0,C 180,E1 -15740.459,E2 -15740.459} C_VEL
LIN {X 0,Y 203.952,Z 902.721,A -85,B 0,C 180,E1 -15745.784,E2 -15745.784} C_VEL
LIN {X 0,Y 203.71,Z 903.203,A -85,B 0,C 180,E1 -15751.126,E2 -15751.126} C_VEL
LIN {X 0,Y 204.327,Z 902.034,A -85,B 0,C 180,E1 -15756.598,E2 -15756.598} C_VEL
LIN {X 0,Y 205.921,Z 899.13,A -85,B 0,C 180,E1 -15762.052,E2 -15762.052} C_VEL
LIN {X 0,Y 208.438,Z 894.796,A -85,B 0,C 180,E1 -15767.015,E2 -15767.015} C_VEL
LIN {X 0,Y 212.06,Z 888.742,A -85,B 0,C 180,E1 -15771.87,E2 -15771.87} C_VEL
LIN {X 0,Y 216.601,Z 881.074,A -85,B 0,C 180,E1 -15776.422,E2 -15776.422} C_VEL
LIN {X 0,Y 221.924,Z 871.794,A -85,B 0,C 180,E1 -15780.622,E2 -15780.622} C_VEL
LIN {X 0,Y 227.869,Z 860.826,A -85,B 0,C 180,E1 -15784.475,E2 -15784.475} C_VEL
LIN {X 0,Y 234.141,Z 848.178,A -85,B 0,C 180,E1 -15787.948,E2 -15787.948} C_VEL
LIN {X 0,Y 240.234,Z 834.497,A -85,B 0,C 180,E1 -15790.907,E2 -15790.907} C_VEL
LIN {X 0,Y 245.919,Z 820.007,A -85,B 0,C 180,E1 -15793.404,E2 -15793.404} C_VEL
LIN {X 0,Y 251.235,Z 804.067,A -85,B 0,C 180,E1 -15795.593,E2 -15795.593} C_VEL
LIN {X 0,Y 255.671,Z 788.092,A -85,B 0,C 180,E1 -15797.327,E2 -15797.327} C_VEL
LIN {X 0,Y 259.416,Z 771.079,A -85,B 0,C 180,E1 -15798.769,E2 -15798.769} C_VEL
LIN {X 0,Y 262.321,Z 752.761,A -85,B 0,C 180,E1 -15799.946,E2 -15799.946} C_VEL
LIN {X 0,Y 263.691,Z 739.018,A -85,B 0,C 180,E1 -15800.64,E2 -15800.64} C_VEL
LIN {X 0,Y 259.912,Z 745.464,A -85,B 0,C 180,E1 -15801.255,E2 -15801.255} C_VEL
LIN {X 0,Y 259.544,Z 746.509,A -85,B 0,C 180,E1 -15801.285,E2 -15801.285} C_VEL
LIN {X 0,Y 258.181,Z 751.701,A -85,B 0,C 180,E1 -15801.257,E2 -15801.257} C_VEL
LIN {X 0,Y 255.816,Z 764.238,A -85,B 0,C 180,E1 -15800.659,E2 -15800.659} C_VEL
LIN {X 0,Y 253.835,Z 768.973,A -85,B 0,C 180,E1 -15800.68,E2 -15800.68} C_VEL
LIN {X 0,Y 253.457,Z 769.583,A -85,B 0,C 180,E1 -15800.714,E2 -15800.714} C_VEL
LIN {X 0,Y 248.121,Z 776.734,A -85,B 0,C 180,E1 -15801.424,E2 -15801.424} C_VEL
LIN {X 0,Y 245.307,Z 779.753,A -85,B 0,C 180,E1 -15801.876,E2 -15801.876} C_VEL
LIN {X 0,Y 240.513,Z 786.874,A -85,B 0,C 180,E1 -15802.329,E2 -15802.329} C_VEL
LIN {X 0,Y 235.885,Z 792.099,A -85,B 0,C 180,E1 -15802.993,E2 -15802.993} C_VEL
LIN {X 0,Y 231.42,Z 796.053,A -85,B 0,C 180,E1 -15803.897,E2 -15803.897} C_VEL
LIN {X 0,Y 227.119,Z 801.002,A -85,B 0,C 180,E1 -15804.47,E2 -15804.47} C_VEL
LIN {X 0,Y 223.072,Z 804.609,A -85,B 0,C 180,E1 -15805.302,E2 -15805.302} C_VEL
LIN {X 0,Y 220.335,Z 806.387,A -85,B 0,C 180,E1 -15806.07,E2 -15806.07} C_VEL
LIN {X 0,Y 216.454,Z 810.354,A -85,B 0,C 180,E1 -15806.731,E2 -15806.731} C_VEL
LIN {X 0,Y 213.095,Z 812.75,A -85,B 0,C 180,E1 -15807.662,E2 -15807.662} C_VEL
LIN {X 0,Y 211.589,Z 813.082,A -85,B 0,C 180,E1 -15808.363,E2 -15808.363} C_VEL
LIN {X 0,Y 208.718,Z 828.877,A -85,B 0,C 180,E1 -15810.749,E2 -15810.749} C_VEL
LIN {X 0,Y 205.46,Z 845.229,A -85,B 0,C 180,E1 -15813.869,E2 -15813.869} C_VEL
LIN {X 0,Y 202.237,Z 860.656,A -85,B 0,C 180,E1 -15817.623,E2 -15817.623} C_VEL
LIN {X 0,Y 199.609,Z 873.721,A -85,B 0,C 180,E1 -15821.604,E2 -15821.604} C_VEL
LIN {X 0,Y 197.7,Z 884.49,A -85,B 0,C 180,E1 -15825.651,E2 -15825.651} C_VEL
LIN {X 0,Y 196.311,Z 895.031,A -85,B 0,C 180,E1 -15830.619,E2 -15830.619} C_VEL
LIN {X 0,Y 195.894,Z 903.259,A -85,B 0,C 180,E1 -15835.608,E2 -15835.608} C_VEL
LIN {X 0,Y 196.407,Z 909.539,A -85,B 0,C 180,E1 -15840.583,E2 -15840.583} C_VEL
LIN {X 0,Y 198.018,Z 914.348,A -85,B 0,C 180,E1 -15845.795,E2 -15845.795} C_VEL
LIN {X 0,Y 201.283,Z 917.591,A -85,B 0,C 180,E1 -15851.46,E2 -15851.46} C_VEL
LIN {X 0,Y 206.545,Z 918.8,A -85,B 0,C 180,E1 -15857.174,E2 -15857.174} C_VEL
LIN {X 0,Y 213.767,Z 917.944,A -85,B 0,C 180,E1 -15862.552,E2 -15862.552} C_VEL
LIN {X 0,Y 222.883,Z 915.178,A -85,B 0,C 180,E1 -15867.519,E2 -15867.519} C_VEL
LIN {X 0,Y 234.481,Z 910.428,A -85,B 0,C 180,E1 -15872.209,E2 -15872.209} C_VEL
LIN {X 0,Y 246.575,Z 904.723,A -85,B 0,C 180,E1 -15875.954,E2 -15875.954} C_VEL
LIN {X 0,Y 228.912,Z 919.186,A -85,B 0,C 180,E1 -15881.298,E2 -15881.298} C_VEL
LIN {X 0,Y 213.547,Z 933.831,A -85,B 0,C 180,E1 -15888.327,E2 -15888.327} C_VEL
LIN {X 0,Y 202.562,Z 946.728,A -85,B 0,C 180,E1 -15896.437,E2 -15896.437} C_VEL
LIN {X 0,Y 196.508,Z 956.244,A -85,B 0,C 180,E1 -15904.373,E2 -15904.373} C_VEL
LIN {X 0,Y 194.02,Z 962.56,A -85,B 0,C 180,E1 -15911.479,E2 -15911.479} C_VEL
LIN {X 0,Y 193.612,Z 966.622,A -85,B 0,C 180,E1 -15918.078,E2 -15918.078} C_VEL
LIN {X 0,Y 194.175,Z 968.547,A -85,B 0,C 180,E1 -15923.614,E2 -15923.614} C_VEL
LIN {X 0,Y 194.731,Z 968.89,A -85,B 0,C 180,E1 -15927.939,E2 -15927.939} C_VEL
LIN {X 0,Y 194.884,Z 968.133,A -85,B 0,C 180,E1 -15932.057,E2 -15932.057} C_VEL
LIN {X 0,Y 194.593,Z 966.044,A -85,B 0,C 180,E1 -15936.49,E2 -15936.49} C_VEL
LIN {X 0,Y 194.211,Z 961.803,A -85,B 0,C 180,E1 -15942.487,E2 -15942.487} C_VEL
LIN {X 0,Y 194.566,Z 956.455,A -85,B 0,C 180,E1 -15947.958,E2 -15947.958} C_VEL
LIN {X 0,Y 196.067,Z 949.212,A -85,B 0,C 180,E1 -15953.438,E2 -15953.438} C_VEL
LIN {X 0,Y 198.675,Z 940.471,A -85,B 0,C 180,E1 -15958.56,E2 -15958.56} C_VEL
LIN {X 0,Y 202.387,Z 930.071,A -85,B 0,C 180,E1 -15963.395,E2 -15963.395} C_VEL
LIN {X 0,Y 207.019,Z 918.122,A -85,B 0,C 180,E1 -15967.834,E2 -15967.834} C_VEL
LIN {X 0,Y 212.22,Z 904.96,A -85,B 0,C 180,E1 -15971.754,E2 -15971.754} C_VEL
LIN {X 0,Y 217.644,Z 890.642,A -85,B 0,C 180,E1 -15975.195,E2 -15975.195} C_VEL
LIN {X 0,Y 223.284,Z 875.006,A -85,B 0,C 180,E1 -15978.189,E2 -15978.189} C_VEL
LIN {X 0,Y 228.562,Z 858.399,A -85,B 0,C 180,E1 -15980.74,E2 -15980.74} C_VEL
LIN {X 0,Y 232.967,Z 843.98,A -85,B 0,C 180,E1 -15982.559,E2 -15982.559} C_VEL
LIN {X 0,Y 240.362,Z 822.159,A -85,B 0,C 180,E1 -15985.298,E2 -15985.298} C_VEL
LIN {X 0,Y 247.503,Z 799.154,A -85,B 0,C 180,E1 -15987.598,E2 -15987.598} C_VEL
LIN {X 0,Y 254.221,Z 775.06,A -85,B 0,C 180,E1 -15989.465,E2 -15989.465} C_VEL
LIN {X 0,Y 259.999,Z 750.54,A -85,B 0,C 180,E1 -15990.921,E2 -15990.921} C_VEL
LIN {X 0,Y 264.395,Z 725.859,A -85,B 0,C 180,E1 -15992.053,E2 -15992.053} C_VEL
LIN {X 0,Y 269.409,Z 698.827,A -85,B 0,C 180,E1 -15992.816,E2 -15992.816} C_VEL
LIN {X 0,Y 271.077,Z 691.126,A -85,B 0,C 180,E1 -15992.968,E2 -15992.968} C_VEL
LIN {X 0,Y 283.55,Z 667.05,A -85,B 0,C 180,E1 -15994.282,E2 -15994.282} C_VEL
LIN {X 0,Y 288.83,Z 656.916,A -85,B 0,C 180,E1 -15994.8,E2 -15994.8} C_VEL
LIN {X 0,Y 287.452,Z 633.553,A -85,B 0,C 180,E1 -15998.472,E2 -15998.472} C_VEL
LIN {X 0,Y 288.689,Z 609.467,A -85,B 0,C 180,E1 -16001.943,E2 -16001.943} C_VEL
LIN {X 0,Y 292.51,Z 583.458,A -85,B 0,C 180,E1 -16005.317,E2 -16005.317} C_VEL
LIN {X 0,Y 293.085,Z 579.902,A -85,B 0,C 180,E1 -16005.782,E2 -16005.782} C_VEL
LIN {X 0,Y 285.743,Z 565.078,A -85,B 0,C 180,E1 -16010.128,E2 -16010.128} C_VEL
LIN {X 0,Y 279.023,Z 551.75,A -85,B 0,C 180,E1 -16014.448,E2 -16014.448} C_VEL
LIN {X 0,Y 271.979,Z 538.261,A -85,B 0,C 180,E1 -16019.314,E2 -16019.314} C_VEL
LIN {X 0,Y 265.315,Z 525.729,A -85,B 0,C 180,E1 -16024.323,E2 -16024.323} C_VEL
LIN {X 0,Y 259.433,Z 515.12,A -85,B 0,C 180,E1 -16029.092,E2 -16029.092} C_VEL
LIN {X 0,Y 254.698,Z 506.321,A -85,B 0,C 180,E1 -16033.393,E2 -16033.393} C_VEL
LIN {X 0,Y 251.763,Z 500.845,A -85,B 0,C 180,E1 -16036.379,E2 -16036.379} C_VEL
LIN {X 0,Y 259.593,Z 498.174,A -85,B 0,C 180,E1 -16041.464,E2 -16041.464} C_VEL
LIN {X 0,Y 261.793,Z 497.836,A -85,B 0,C 180,E1 -16042.691,E2 -16042.691} C_VEL
LIN {X 0,Y 265.956,Z 508.72,A -85,B 0,C 180,E1 -16046.817,E2 -16046.817} C_VEL
LIN {X 0,Y 270.007,Z 520.812,A -85,B 0,C 180,E1 -16050.486,E2 -16050.486} C_VEL
LIN {X 0,Y 272.444,Z 528.286,A -85,B 0,C 180,E1 -16052.369,E2 -16052.369} C_VEL
LIN {X 0,Y 273.449,Z 530.916,A -85,B 0,C 180,E1 -16052.841,E2 -16052.841} C_VEL
LIN {X 0,Y 273.401,Z 535.606,A -85,B 0,C 180,E1 -16053.054,E2 -16053.054} C_VEL
LIN {X 0,Y 260.109,Z 716.74,A -85,B 0,C 180,E1 -16057.366,E2 -16057.366} C_VEL
LIN {X 0,Y 258.588,Z 741.241,A -85,B 0,C 180,E1 -16058.195,E2 -16058.195} C_VEL
LIN {X 0,Y 256.333,Z 759.753,A -85,B 0,C 180,E1 -16059.155,E2 -16059.155} C_VEL
LIN {X 0,Y 253.194,Z 776.893,A -85,B 0,C 180,E1 -16060.364,E2 -16060.364} C_VEL
LIN {X 0,Y 249.119,Z 793.541,A -85,B 0,C 180,E1 -16061.883,E2 -16061.883} C_VEL
LIN {X 0,Y 244.097,Z 810.013,A -85,B 0,C 180,E1 -16063.809,E2 -16063.809} C_VEL
LIN {X 0,Y 238.533,Z 825.3,A -85,B 0,C 180,E1 -16066.075,E2 -16066.075} C_VEL
LIN {X 0,Y 232.294,Z 839.97,A -85,B 0,C 180,E1 -16068.811,E2 -16068.811} C_VEL
LIN {X 0,Y 225.7,Z 853.648,A -85,B 0,C 180,E1 -16072.051,E2 -16072.051} C_VEL
LIN {X 0,Y 219.428,Z 865.407,A -85,B 0,C 180,E1 -16075.597,E2 -16075.597} C_VEL
LIN {X 0,Y 213.417,Z 875.813,A -85,B 0,C 180,E1 -16079.604,E2 -16079.604} C_VEL
LIN {X 0,Y 207.994,Z 884.719,A -85,B 0,C 180,E1 -16084.059,E2 -16084.059} C_VEL
LIN {X 0,Y 203.375,Z 892.098,A -85,B 0,C 180,E1 -16088.969,E2 -16088.969} C_VEL
LIN {X 0,Y 199.738,Z 897.855,A -85,B 0,C 180,E1 -16094.318,E2 -16094.318} C_VEL
LIN {X 0,Y 197.369,Z 901.741,A -85,B 0,C 180,E1 -16099.788,E2 -16099.788} C_VEL
LIN {X 0,Y 196.111,Z 903.924,A -85,B 0,C 180,E1 -16105.322,E2 -16105.322} C_VEL
LIN {X 0,Y 195.805,Z 904.487,A -85,B 0,C 180,E1 -16110.879,E2 -16110.879} C_VEL
LIN {X 0,Y 196.39,Z 903.451,A -85,B 0,C 180,E1 -16116.432,E2 -16116.432} C_VEL
LIN {X 0,Y 197.955,Z 900.774,A -85,B 0,C 180,E1 -16121.953,E2 -16121.953} C_VEL
LIN {X 0,Y 200.694,Z 896.342,A -85,B 0,C 180,E1 -16127.394,E2 -16127.394} C_VEL
LIN {X 0,Y 204.553,Z 890.27,A -85,B 0,C 180,E1 -16132.505,E2 -16132.505} C_VEL
LIN {X 0,Y 209.411,Z 882.528,A -85,B 0,C 180,E1 -16137.283,E2 -16137.283} C_VEL
LIN {X 0,Y 214.758,Z 873.689,A -85,B 0,C 180,E1 -16141.43,E2 -16141.43} C_VEL
LIN {X 0,Y 220.969,Z 862.817,A -85,B 0,C 180,E1 -16145.394,E2 -16145.394} C_VEL
LIN {X 0,Y 227.496,Z 850.362,A -85,B 0,C 180,E1 -16148.94,E2 -16148.94} C_VEL
LIN {X 0,Y 233.885,Z 836.771,A -85,B 0,C 180,E1 -16151.977,E2 -16151.977} C_VEL
LIN {X 0,Y 239.955,Z 822.027,A -85,B 0,C 180,E1 -16154.581,E2 -16154.581} C_VEL
LIN {X 0,Y 245.503,Z 806.169,A -85,B 0,C 180,E1 -16156.805,E2 -16156.805} C_VEL
LIN {X 0,Y 250.112,Z 790.405,A -85,B 0,C 180,E1 -16158.553,E2 -16158.553} C_VEL
LIN {X 0,Y 254.075,Z 773.346,A -85,B 0,C 180,E1 -16160.033,E2 -16160.033} C_VEL
LIN {X 0,Y 255.257,Z 766.757,A -85,B 0,C 180,E1 -16160.535,E2 -16160.535} C_VEL
LIN {X 0,Y 253.457,Z 769.583,A -85,B 0,C 180,E1 -16160.714,E2 -16160.714} C_VEL
LIN {X 0,Y 250.649,Z 774.86,A -85,B 0,C 180,E1 -16160.884,E2 -16160.884} C_VEL
LIN {X 0,Y 245.114,Z 787.312,A -85,B 0,C 180,E1 -16160.672,E2 -16160.672} C_VEL
LIN {X 0,Y 242.685,Z 791.026,A -85,B 0,C 180,E1 -16160.794,E2 -16160.794} C_VEL
LIN {X 0,Y 237.462,Z 796.763,A -85,B 0,C 180,E1 -16161.451,E2 -16161.451} C_VEL
LIN {X 0,Y 232.385,Z 801.15,A -85,B 0,C 180,E1 -16162.34,E2 -16162.34} C_VEL
LIN {X 0,Y 227.476,Z 806.38,A -85,B 0,C 180,E1 -16162.973,E2 -16162.973} C_VEL
LIN {X 0,Y 222.45,Z 810.526,A -85,B 0,C 180,E1 -16163.926,E2 -16163.926} C_VEL
LIN {X 0,Y 220.275,Z 811.917,A -85,B 0,C 180,E1 -16164.477,E2 -16164.477} C_VEL
LIN {X 0,Y 215.778,Z 816.083,A -85,B 0,C 180,E1 -16165.252,E2 -16165.252} C_VEL
LIN {X 0,Y 212.03,Z 818.674,A -85,B 0,C 180,E1 -16166.189,E2 -16166.189} C_VEL
LIN {X 0,Y 210.154,Z 819.569,A -85,B 0,C 180,E1 -16166.828,E2 -16166.828} C_VEL
LIN {X 0,Y 205.947,Z 823.218,A -85,B 0,C 180,E1 -16167.72,E2 -16167.72} C_VEL
LIN {X 0,Y 203.339,Z 824.783,A -85,B 0,C 180,E1 -16168.585,E2 -16168.585} C_VEL
LIN {X 0,Y 202.034,Z 825.017,A -85,B 0,C 180,E1 -16169.27,E2 -16169.27} C_VEL
LIN {X 0,Y 198.669,Z 841.597,A -85,B 0,C 180,E1 -16172.349,E2 -16172.349} C_VEL
LIN {X 0,Y 195.337,Z 857.125,A -85,B 0,C 180,E1 -16175.987,E2 -16175.987} C_VEL
LIN {X 0,Y 192.487,Z 870.592,A -85,B 0,C 180,E1 -16179.95,E2 -16179.95} C_VEL
LIN {X 0,Y 190.275,Z 882.097,A -85,B 0,C 180,E1 -16184.141,E2 -16184.141} C_VEL
LIN {X 0,Y 188.65,Z 892.878,A -85,B 0,C 180,E1 -16188.999,E2 -16188.999} C_VEL
LIN {X 0,Y 187.938,Z 901.896,A -85,B 0,C 180,E1 -16194.201,E2 -16194.201} C_VEL
LIN {X 0,Y 188.18,Z 908.568,A -85,B 0,C 180,E1 -16199.086,E2 -16199.086} C_VEL
LIN {X 0,Y 189.643,Z 914.447,A -85,B 0,C 180,E1 -16204.838,E2 -16204.838} C_VEL
LIN {X 0,Y 192.742,Z 918.48,A -85,B 0,C 180,E1 -16210.762,E2 -16210.762} C_VEL
LIN {X 0,Y 197.915,Z 920.515,A -85,B 0,C 180,E1 -16216.735,E2 -16216.735} C_VEL
LIN {X 0,Y 205.116,Z 920.493,A -85,B 0,C 180,E1 -16222.346,E2 -16222.346} C_VEL
LIN {X 0,Y 214.783,Z 918.473,A -85,B 0,C 180,E1 -16227.743,E2 -16227.743} C_VEL
LIN {X 0,Y 226.569,Z 914.57,A -85,B 0,C 180,E1 -16232.573,E2 -16232.573} C_VEL
LIN {X 0,Y 236.734,Z 910.579,A -85,B 0,C 180,E1 -16235.813,E2 -16235.813} C_VEL
LIN {X 0,Y 218.957,Z 924.056,A -85,B 0,C 180,E1 -16241.504,E2 -16241.504} C_VEL
LIN {X 0,Y 203.385,Z 937.917,A -85,B 0,C 180,E1 -16249.206,E2 -16249.206} C_VEL
LIN {X 0,Y 193.556,Z 948.748,A -85,B 0,C 180,E1 -16257.152,E2 -16257.152} C_VEL
LIN {X 0,Y 188.035,Z 957.032,A -85,B 0,C 180,E1 -16265.16,E2 -16265.16} C_VEL
LIN {X 0,Y 185.9,Z 962.505,A -85,B 0,C 180,E1 -16272.47,E2 -16272.47} C_VEL
LIN {X 0,Y 185.77,Z 965.837,A -85,B 0,C 180,E1 -16279.141,E2 -16279.141} C_VEL
LIN {X 0,Y 186.438,Z 967.153,A -85,B 0,C 180,E1 -16284.46,E2 -16284.46} C_VEL
LIN {X 0,Y 187,Z 967.124,A -85,B 0,C 180,E1 -16288.988,E2 -16288.988} C_VEL
LIN {X 0,Y 187.035,Z 966.039,A -85,B 0,C 180,E1 -16293.064,E2 -16293.064} C_VEL
LIN {X 0,Y 186.531,Z 963.573,A -85,B 0,C 180,E1 -16298.321,E2 -16298.321} C_VEL
LIN {X 0,Y 186.244,Z 959.994,A -85,B 0,C 180,E1 -16303.666,E2 -16303.666} C_VEL
LIN {X 0,Y 186.771,Z 954.785,A -85,B 0,C 180,E1 -16309.059,E2 -16309.059} C_VEL
LIN {X 0,Y 188.555,Z 947.421,A -85,B 0,C 180,E1 -16314.765,E2 -16314.765} C_VEL
LIN {X 0,Y 191.534,Z 938.56,A -85,B 0,C 180,E1 -16320.075,E2 -16320.075} C_VEL
LIN {X 0,Y 195.56,Z 928.318,A -85,B 0,C 180,E1 -16324.933,E2 -16324.933} C_VEL
LIN {X 0,Y 200.767,Z 915.949,A -85,B 0,C 180,E1 -16329.602,E2 -16329.602} C_VEL
LIN {X 0,Y 206.671,Z 901.98,A -85,B 0,C 180,E1 -16333.773,E2 -16333.773} C_VEL
LIN {X 0,Y 212.772,Z 886.839,A -85,B 0,C 180,E1 -16337.342,E2 -16337.342} C_VEL
LIN {X 0,Y 218.827,Z 870.672,A -85,B 0,C 180,E1 -16340.344,E2 -16340.344} C_VEL
LIN {X 0,Y 224.233,Z 854.408,A -85,B 0,C 180,E1 -16342.743,E2 -16342.743} C_VEL
LIN {X 0,Y 229.155,Z 837.237,A -85,B 0,C 180,E1 -16344.74,E2 -16344.74} C_VEL
LIN {X 0,Y 232.724,Z 823.792,A -85,B 0,C 180,E1 -16346.015,E2 -16346.015} C_VEL
LIN {X 0,Y 240.071,Z 801.008,A -85,B 0,C 180,E1 -16348.397,E2 -16348.397} C_VEL
LIN {X 0,Y 246.803,Z 777.898,A -85,B 0,C 180,E1 -16350.29,E2 -16350.29} C_VEL
LIN {X 0,Y 252.891,Z 753.682,A -85,B 0,C 180,E1 -16351.814,E2 -16351.814} C_VEL
LIN {X 0,Y 257.613,Z 729.086,A -85,B 0,C 180,E1 -16353.027,E2 -16353.027} C_VEL
LIN {X 0,Y 262.343,Z 703.248,A -85,B 0,C 180,E1 -16353.822,E2 -16353.822} C_VEL
LIN {X 0,Y 265.305,Z 690.021,A -85,B 0,C 180,E1 -16354.128,E2 -16354.128} C_VEL
LIN {X 0,Y 278.112,Z 665.646,A -85,B 0,C 180,E1 -16355.446,E2 -16355.446} C_VEL
LIN {X 0,Y 282.132,Z 658.045,A -85,B 0,C 180,E1 -16355.832,E2 -16355.832} C_VEL
LIN {X 0,Y 281.132,Z 634.227,A -85,B 0,C 180,E1 -16359.603,E2 -16359.603} C_VEL
LIN {X 0,Y 282.793,Z 609.742,A -85,B 0,C 180,E1 -16363.147,E2 -16363.147} C_VEL
LIN {X 0,Y 286.827,Z 583.904,A -85,B 0,C 180,E1 -16366.548,E2 -16366.548} C_VEL
LIN {X 0,Y 279.259,Z 568.47,A -85,B 0,C 180,E1 -16371.183,E2 -16371.183} C_VEL
LIN {X 0,Y 272.548,Z 555.273,A -85,B 0,C 180,E1 -16375.582,E2 -16375.582} C_VEL
LIN {X 0,Y 266.001,Z 542.689,A -85,B 0,C 180,E1 -16380.216,E2 -16380.216} C_VEL
LIN {X 0,Y 259.727,Z 530.797,A -85,B 0,C 180,E1 -16385.08,E2 -16385.08} C_VEL
LIN {X 0,Y 253.841,Z 519.998,A -85,B 0,C 180,E1 -16390.029,E2 -16390.029} C_VEL
LIN {X 0,Y 249.089,Z 511.189,A -85,B 0,C 180,E1 -16394.411,E2 -16394.411} C_VEL
LIN {X 0,Y 248.233,Z 509.138,A -85,B 0,C 180,E1 -16395.537,E2 -16395.537} C_VEL
LIN {X 0,Y 256.647,Z 505.924,A -85,B 0,C 180,E1 -16401.243,E2 -16401.243} C_VEL
LIN {X 0,Y 258.827,Z 505.714,A -85,B 0,C 180,E1 -16402.546,E2 -16402.546} C_VEL
LIN {X 0,Y 262.604,Z 516.025,A -85,B 0,C 180,E1 -16406.454,E2 -16406.454} C_VEL
LIN {X 0,Y 266.545,Z 528.618,A -85,B 0,C 180,E1 -16410.239,E2 -16410.239} C_VEL
LIN {X 0,Y 269.285,Z 535.017,A -85,B 0,C 180,E1 -16411.595,E2 -16411.595} C_VEL
LIN {X 0,Y 255.412,Z 717.19,A -85,B 0,C 180,E1 -16415.93,E2 -16415.93} C_VEL
LIN {X 0,Y 253.776,Z 742.366,A -85,B 0,C 180,E1 -16416.786,E2 -16416.786} C_VEL
LIN {X 0,Y 251.419,Z 760.944,A -85,B 0,C 180,E1 -16417.754,E2 -16417.754} C_VEL
LIN {X 0,Y 248.177,Z 778.01,A -85,B 0,C 180,E1 -16418.963,E2 -16418.963} C_VEL
LIN {X 0,Y 243.914,Z 794.789,A -85,B 0,C 180,E1 -16420.501,E2 -16420.501} C_VEL
LIN {X 0,Y 238.897,Z 810.704,A -85,B 0,C 180,E1 -16422.365,E2 -16422.365} C_VEL
LIN {X 0,Y 233.173,Z 825.917,A -85,B 0,C 180,E1 -16424.618,E2 -16424.618} C_VEL
LIN {X 0,Y 226.913,Z 840.168,A -85,B 0,C 180,E1 -16427.268,E2 -16427.268} C_VEL
LIN {X 0,Y 220.539,Z 852.986,A -85,B 0,C 180,E1 -16430.265,E2 -16430.265} C_VEL
LIN {X 0,Y 213.79,Z 865.208,A -85,B 0,C 180,E1 -16433.895,E2 -16433.895} C_VEL
LIN {X 0,Y 207.364,Z 875.878,A -85,B 0,C 180,E1 -16437.969,E2 -16437.969} C_VEL
LIN {X 0,Y 201.513,Z 885.018,A -85,B 0,C 180,E1 -16442.521,E2 -16442.521} C_VEL
LIN {X 0,Y 196.48,Z 892.609,A -85,B 0,C 180,E1 -16447.564,E2 -16447.564} C_VEL
LIN {X 0,Y 192.641,Z 898.321,A -85,B 0,C 180,E1 -16452.793,E2 -16452.793} C_VEL
LIN {X 0,Y 189.903,Z 902.517,A -85,B 0,C 180,E1 -16458.46,E2 -16458.46} C_VEL
LIN {X 0,Y 188.384,Z 904.976,A -85,B 0,C 180,E1 -16464.213,E2 -16464.213} C_VEL
LIN {X 0,Y 187.901,Z 905.802,A -85,B 0,C 180,E1 -16470.001,E2 -16470.001} C_VEL
LIN {X 0,Y 188.373,Z 905.024,A -85,B 0,C 180,E1 -16475.789,E2 -16475.789} C_VEL
LIN {X 0,Y 189.878,Z 902.608,A -85,B 0,C 180,E1 -16481.544,E2 -16481.544} C_VEL
LIN {X 0,Y 192.599,Z 898.45,A -85,B 0,C 180,E1 -16487.213,E2 -16487.213} C_VEL
LIN {X 0,Y 196.423,Z 892.783,A -85,B 0,C 180,E1 -16492.445,E2 -16492.445} C_VEL
LIN {X 0,Y 201.135,Z 885.725,A -85,B 0,C 180,E1 -16497.217,E2 -16497.217} C_VEL
LIN {X 0,Y 206.912,Z 876.753,A -85,B 0,C 180,E1 -16501.785,E2 -16501.785} C_VEL
LIN {X 0,Y 213.275,Z 866.27,A -85,B 0,C 180,E1 -16505.876,E2 -16505.876} C_VEL
LIN {X 0,Y 219.971,Z 854.266,A -85,B 0,C 180,E1 -16509.522,E2 -16509.522} C_VEL
LIN {X 0,Y 226.809,Z 840.641,A -85,B 0,C 180,E1 -16512.758,E2 -16512.758} C_VEL
LIN {X 0,Y 233.069,Z 826.479,A -85,B 0,C 180,E1 -16515.41,E2 -16515.41} C_VEL
LIN {X 0,Y 238.77,Z 811.448,A -85,B 0,C 180,E1 -16517.656,E2 -16517.656} C_VEL
LIN {X 0,Y 243.81,Z 795.628,A -85,B 0,C 180,E1 -16519.53,E2 -16519.53} C_VEL
LIN {X 0,Y 246.276,Z 786.243,A -85,B 0,C 180,E1 -16520.479,E2 -16520.479} C_VEL
LIN {X 0,Y 242.685,Z 791.026,A -85,B 0,C 180,E1 -16520.794,E2 -16520.794} C_VEL
LIN {X 0,Y 238.862,Z 796.607,A -85,B 0,C 180,E1 -16520.999,E2 -16520.999} C_VEL
LIN {X 0,Y 232.302,Z 806.803,A -85,B 0,C 180,E1 -16521.01,E2 -16521.01} C_VEL
LIN {X 0,Y 228.962,Z 810.608,A -85,B 0,C 180,E1 -16521.294,E2 -16521.294} C_VEL
LIN {X 0,Y 223.421,Z 815.16,A -85,B 0,C 180,E1 -16522.185,E2 -16522.185} C_VEL
LIN {X 0,Y 219.348,Z 818.033,A -85,B 0,C 180,E1 -16523.007,E2 -16523.007} C_VEL
LIN {X 0,Y 213.854,Z 822.539,A -85,B 0,C 180,E1 -16523.985,E2 -16523.985} C_VEL
LIN {X 0,Y 208.9,Z 825.46,A -85,B 0,C 180,E1 -16525.279,E2 -16525.279} C_VEL
LIN {X 0,Y 203.893,Z 829.275,A -85,B 0,C 180,E1 -16526.348,E2 -16526.348} C_VEL
LIN {X 0,Y 200.006,Z 831.293,A -85,B 0,C 180,E1 -16527.661,E2 -16527.661} C_VEL
LIN {X 0,Y 195.446,Z 834.577,A -85,B 0,C 180,E1 -16528.888,E2 -16528.888} C_VEL
LIN {X 0,Y 193.146,Z 835.61,A -85,B 0,C 180,E1 -16529.857,E2 -16529.857} C_VEL
LIN {X 0,Y 192.42,Z 835.69,A -85,B 0,C 180,E1 -16530.333,E2 -16530.333} C_VEL
LIN {X 0,Y 189.123,Z 850.776,A -85,B 0,C 180,E1 -16533.634,E2 -16533.634} C_VEL
LIN {X 0,Y 185.934,Z 865.064,A -85,B 0,C 180,E1 -16537.554,E2 -16537.554} C_VEL
LIN {X 0,Y 183.282,Z 877.791,A -85,B 0,C 180,E1 -16541.882,E2 -16541.882} C_VEL
LIN {X 0,Y 181.404,Z 888.261,A -85,B 0,C 180,E1 -16546.289,E2 -16546.289} C_VEL
LIN {X 0,Y 180.207,Z 898.076,A -85,B 0,C 180,E1 -16551.383,E2 -16551.383} C_VEL
LIN {X 0,Y 179.984,Z 906.305,A -85,B 0,C 180,E1 -16556.815,E2 -16556.815} C_VEL
LIN {X 0,Y 180.822,Z 912.671,A -85,B 0,C 180,E1 -16562.217,E2 -16562.217} C_VEL
LIN {X 0,Y 183.134,Z 917.827,A -85,B 0,C 180,E1 -16568.16,E2 -16568.16} C_VEL
LIN {X 0,Y 187.324,Z 921.211,A -85,B 0,C 180,E1 -16574.212,E2 -16574.212} C_VEL
LIN {X 0,Y 193.795,Z 922.678,A -85,B 0,C 180,E1 -16580.222,E2 -16580.222} C_VEL
LIN {X 0,Y 202.796,Z 922.172,A -85,B 0,C 180,E1 -16586.027,E2 -16586.027} C_VEL
LIN {X 0,Y 214.565,Z 919.596,A -85,B 0,C 180,E1 -16591.46,E2 -16591.46} C_VEL
LIN {X 0,Y 226.757,Z 915.866,A -85,B 0,C 180,E1 -16595.675,E2 -16595.675} C_VEL
LIN {X 0,Y 207.86,Z 929.206,A -85,B 0,C 180,E1 -16602.201,E2 -16602.201} C_VEL
LIN {X 0,Y 192.526,Z 942.049,A -85,B 0,C 180,E1 -16610.683,E2 -16610.683} C_VEL
LIN {X 0,Y 183.544,Z 951.671,A -85,B 0,C 180,E1 -16619.197,E2 -16619.197} C_VEL
LIN {X 0,Y 178.997,Z 958.674,A -85,B 0,C 180,E1 -16627.675,E2 -16627.675} C_VEL
LIN {X 0,Y 177.73,Z 962.917,A -85,B 0,C 180,E1 -16635.001,E2 -16635.001} C_VEL
LIN {X 0,Y 178.104,Z 965.065,A -85,B 0,C 180,E1 -16641.281,E2 -16641.281} C_VEL
LIN {X 0,Y 178.899,Z 965.638,A -85,B 0,C 180,E1 -16646.474,E2 -16646.474} C_VEL
LIN {X 0,Y 179.28,Z 965.049,A -85,B 0,C 180,E1 -16650.638,E2 -16650.638} C_VEL
LIN {X 0,Y 179.041,Z 963.806,A -85,B 0,C 180,E1 -16654.804,E2 -16654.804} C_VEL
LIN {X 0,Y 178.448,Z 961.557,A -85,B 0,C 180,E1 -16660.002,E2 -16660.002} C_VEL
LIN {X 0,Y 178.354,Z 957.608,A -85,B 0,C 180,E1 -16665.609,E2 -16665.609} C_VEL
LIN {X 0,Y 179.376,Z 951.615,A -85,B 0,C 180,E1 -16671.585,E2 -16671.585} C_VEL
LIN {X 0,Y 181.628,Z 944.174,A -85,B 0,C 180,E1 -16677.187,E2 -16677.187} C_VEL
LIN {X 0,Y 185.27,Z 934.834,A -85,B 0,C 180,E1 -16682.661,E2 -16682.661} C_VEL
LIN {X 0,Y 189.986,Z 924.085,A -85,B 0,C 180,E1 -16687.624,E2 -16687.624} C_VEL
LIN {X 0,Y 195.744,Z 911.496,A -85,B 0,C 180,E1 -16692.214,E2 -16692.214} C_VEL
LIN {X 0,Y 202.02,Z 897.437,A -85,B 0,C 180,E1 -16696.268,E2 -16696.268} C_VEL
LIN {X 0,Y 208.467,Z 882.335,A -85,B 0,C 180,E1 -16699.693,E2 -16699.693} C_VEL
LIN {X 0,Y 214.635,Z 866.343,A -85,B 0,C 180,E1 -16702.57,E2 -16702.57} C_VEL
LIN {X 0,Y 220.516,Z 849.411,A -85,B 0,C 180,E1 -16704.926,E2 -16704.926} C_VEL
LIN {X 0,Y 225.427,Z 832.363,A -85,B 0,C 180,E1 -16706.81,E2 -16706.81} C_VEL
LIN {X 0,Y 229.683,Z 814.332,A -85,B 0,C 180,E1 -16708.325,E2 -16708.325} C_VEL
LIN {X 0,Y 231.707,Z 805.655,A -85,B 0,C 180,E1 -16708.932,E2 -16708.932} C_VEL
LIN {X 0,Y 238.706,Z 782.791,A -85,B 0,C 180,E1 -16710.957,E2 -16710.957} C_VEL
LIN {X 0,Y 245.161,Z 758.854,A -85,B 0,C 180,E1 -16712.588,E2 -16712.588} C_VEL
LIN {X 0,Y 250.319,Z 734.563,A -85,B 0,C 180,E1 -16713.885,E2 -16713.885} C_VEL
LIN {X 0,Y 254.726,Z 710.632,A -85,B 0,C 180,E1 -16714.774,E2 -16714.774} C_VEL
